C01709=71.781,53.873,81.904,-174.9523,-0.9140,-13823.1111
C01710=77.964,55.051,82.431,-177.5443,-2.1205,-13824.7738
C01711=83.695,52.900,82.857,-179.4162,-1.4469,-13827.7048
C01712=87.788,47.863,83.283,-179.9986,-0.1052,-13831.4003
C01713=90.949,41.570,83.562,-179.9996,-0.0128,-13835.4363
C01714=93.705,34.916,83.562,-179.9986,-0.0127,-13839.5638
C01715=95.920,28.231,83.283,180.0000,-0.1015,-13843.5999
C01716=96.587,21.776,82.857,179.4149,-1.4483,-13847.2948
C01717=94.056,16.202,82.431,177.5455,-2.1207,-13850.2262
C01718=88.851,12.662,81.904,174.9556,-0.9120,-13851.8895
C01719=81.722,11.527,80.892,174.7101,-0.0362,-13851.9713
C01720=73.885,10.553,78.794,175.1749,-0.0294,-13851.8714
C01721=66.709,9.674,75.971,175.9523,-0.0621,-13851.7486
C01722=61.204,8.875,73.167,178.1043,-0.0957,-13851.7492
C01723=57.930,7.507,71.114,-165.0758,11.9424,-13852.6163
C01724=57.039,4.398,70.297,-173.6555,31.1772,-13855.5909
C01725=57.094,1.874,70.261,179.7573,32.5080,-13858.1201
C01726=57.118,0.000,70.285,-180.0000,32.4949,-13860.0000
C01727=57.094,-1.874,70.261,-179.7573,32.5080,-13861.8799
C01728=57.039,-4.398,70.297,173.6555,31.1772,-13864.4091
C01729=57.930,-7.507,71.114,165.0758,11.9424,-13867.3837
C01730=61.204,-8.875,73.167,-178.1043,-0.0957,-13868.2508
C01731=66.709,-9.674,75.971,-175.9523,-0.0621,-13868.2514
C01732=73.885,-10.553,78.794,-175.1749,-0.0294,-13868.1286
C01733=81.722,-11.527,80.892,-174.7101,-0.0362,-13868.0287
C01734=88.851,-12.662,81.904,-174.9556,-0.9120,-13868.1105
C01735=94.056,-16.202,82.431,-177.5455,-2.1207,-13869.7738
C01736=96.587,-21.776,82.857,-179.4149,-1.4483,-13872.7052
C01737=95.920,-28.231,83.283,-180.0000,-0.1015,-13876.4001
C01738=93.705,-34.916,83.562,179.9986,-0.0127,-13880.4362
C01739=90.949,-41.570,83.562,179.9996,-0.0128,-13884.5637
C01740=87.788,-47.863,83.283,179.9986,-0.1052,-13888.5997
C01741=83.695,-52.900,82.857,179.4162,-1.4469,-13892.2952
C01742=77.964,-55.051,82.431,177.5443,-2.1205,-13895.2262
C01743=71.781,-53.873,81.904,174.9523,-0.9140,-13896.8889
C01744=65.937,-49.635,80.892,174.7131,-0.0370,-13896.9711
C01745=59.707,-44.783,78.794,175.1691,-0.0312,-13896.8716
C01746=54.011,-40.330,75.971,175.9514,-0.0603,-13896.7487
C01747=49.553,-37.003,73.167,178.1031,-0.0935,-13896.7500
C01748=46.271,-35.654,71.114,-165.0753,11.9430,-13897.6160
C01749=43.442,-37.223,70.297,-173.6602,31.1794,-13900.5914
C01750=41.697,-39.047,70.261,179.7562,32.5069,-13903.1202
C01751=40.388,-40.388,70.285,-180.0000,32.4978,-13905.0000
C01752=39.047,-41.696,70.261,-179.7558,32.5069,-13906.8791
C01753=37.223,-43.443,70.297,173.6555,31.1756,-13909.4092
C01754=35.654,-46.271,71.114,165.0753,11.9430,-13912.3840
C01755=37.003,-49.553,73.167,-178.1031,-0.0935,-13913.2500
C01756=40.330,-54.011,75.971,-175.9514,-0.0603,-13913.2513
C01757=44.783,-59.707,78.794,-175.1691,-0.0312,-13913.1284
C01758=49.635,-65.937,80.892,-174.7131,-0.0370,-13913.0289
C01759=53.873,-71.781,81.904,-174.9523,-0.9140,-13913.1111
C01760=55.051,-77.964,82.431,-177.5443,-2.1205,-13914.7738
C01761=52.900,-83.695,82.857,-179.4162,-1.4469,-13917.7048
C01762=47.863,-87.788,83.283,-179.9986,-0.1052,-13921.4003
C01763=41.570,-90.949,83.562,-179.9996,-0.0128,-13925.4363
C01764=34.916,-93.705,83.562,-179.9986,-0.0127,-13929.5638
C01765=28.231,-95.920,83.283,180.0000,-0.1015,-13933.5999
C01766=21.776,-96.587,82.857,179.4149,-1.4483,-13937.2948
C01767=16.202,-94.056,82.431,177.5455,-2.1207,-13940.2262
C01768=12.662,-88.851,81.904,174.9556,-0.9120,-13941.8895
C01769=11.527,-81.722,80.892,174.7101,-0.0362,-13941.9713
C01770=10.553,-73.885,78.794,175.1749,-0.0294,-13941.8714
C01771=9.674,-66.709,75.971,175.9523,-0.0621,-13941.7486
C01772=8.875,-61.204,73.167,178.1043,-0.0957,-13941.7492
C01773=7.507,-57.930,71.114,-165.0758,11.9424,-13942.6163
C01774=4.398,-57.039,70.297,-173.6555,31.1772,-13945.5909
C01775=1.874,-57.094,70.261,179.7573,32.5080,-13948.1201
C01776=0.000,-57.118,70.285,-180.0000,32.4949,-13950.0000
C01777=0.000,-57.118,70.285,-180.0000,32.4949,-13950.0000
C01778=-1.874,-57.094,70.261,-179.7573,32.5080,-13951.8799
C01779=-4.398,-57.039,70.297,173.6555,31.1772,-13954.4091
C01780=-7.507,-57.930,71.114,165.0758,11.9424,-13957.3837
C01781=-8.875,-61.204,73.167,-178.1043,-0.0957,-13958.2508
C01782=-9.674,-66.709,75.971,-175.9523,-0.0621,-13958.2514
C01783=-10.553,-73.885,78.794,-175.1749,-0.0294,-13958.1286
C01784=-11.527,-81.722,80.892,-174.7101,-0.0362,-13958.0287
C01785=-12.662,-88.851,81.904,-174.9556,-0.9120,-13958.1105
C01786=-16.202,-94.056,82.431,-177.5455,-2.1207,-13959.7738
C01787=-21.776,-96.587,82.857,-179.4149,-1.4483,-13962.7052
C01788=-28.231,-95.920,83.283,-180.0000,-0.1015,-13966.4001
C01789=-34.916,-93.705,83.562,179.9986,-0.0127,-13970.4362
C01790=-41.570,-90.949,83.562,179.9996,-0.0128,-13974.5637
C01791=-47.863,-87.788,83.283,179.9986,-0.1052,-13978.5997
C01792=-52.900,-83.695,82.857,179.4162,-1.4469,-13982.2952
C01793=-55.051,-77.964,82.431,177.5443,-2.1205,-13985.2262
C01794=-53.873,-71.781,81.904,174.9523,-0.9140,-13986.8889
C01795=-49.635,-65.937,80.892,174.7131,-0.0370,-13986.9711
C01796=-44.783,-59.707,78.794,175.1691,-0.0312,-13986.8716
C01797=-40.330,-54.011,75.971,175.9514,-0.0603,-13986.7487
C01798=-37.003,-49.553,73.167,178.1031,-0.0935,-13986.7500
C01799=-35.654,-46.271,71.114,-165.0753,11.9430,-13987.6160
C01800=-37.223,-43.442,70.297,-173.6602,31.1794,-13990.5914
C01801=-39.047,-41.697,70.261,179.7562,32.5069,-13993.1202
C01802=-40.388,-40.388,70.285,-180.0000,32.4978,-13995.0000
C01803=-41.696,-39.047,70.261,-179.7558,32.5069,-13996.8791
C01804=-43.443,-37.223,70.297,173.6555,31.1756,-13999.4092
C01805=-46.271,-35.654,71.114,165.0753,11.9430,-14002.3840
C01806=-49.553,-37.003,73.167,-178.1031,-0.0935,-14003.2500
C01807=-54.011,-40.330,75.971,-175.9514,-0.0603,-14003.2513
C01808=-59.707,-44.783,78.794,-175.1691,-0.0312,-14003.1284
C01809=-65.937,-49.635,80.892,-174.7131,-0.0370,-14003.0289
C01810=-71.781,-53.873,81.904,-174.9523,-0.9140,-14003.1111
C01811=-77.964,-55.051,82.431,-177.5443,-2.1205,-14004.7738
C01812=-83.695,-52.900,82.857,-179.4162,-1.4469,-14007.7048
C01813=-87.788,-47.863,83.283,-179.9986,-0.1052,-14011.4003
C01814=-90.949,-41.570,83.562,-179.9996,-0.0128,-14015.4363
C01815=-93.705,-34.916,83.562,-179.9986,-0.0127,-14019.5638
C01816=-95.920,-28.231,83.283,180.0000,-0.1015,-14023.5999
C01817=-96.587,-21.776,82.857,179.4149,-1.4483,-14027.2948
C01818=-94.056,-16.202,82.431,177.5455,-2.1207,-14030.2262
C01819=-88.851,-12.662,81.904,174.9556,-0.9120,-14031.8895
C01820=-81.722,-11.527,80.892,174.7101,-0.0362,-14031.9713
C01821=-73.885,-10.553,78.794,175.1749,-0.0294,-14031.8714
C01822=-66.709,-9.674,75.971,175.9523,-0.0621,-14031.7486
C01823=-61.204,-8.875,73.167,178.1043,-0.0957,-14031.7492
C01824=-57.930,-7.507,71.114,-165.0758,11.9424,-14032.6163
C01825=-57.039,-4.398,70.297,-173.6555,31.1772,-14035.5909
C01826=-57.094,-1.874,70.261,179.7573,32.5080,-14038.1201
C01827=-57.118,0.000,70.285,-180.0000,32.4949,-14040.0000
C01828=-57.094,1.874,70.261,-179.7573,32.5080,-14041.8799
C01829=-57.039,4.398,70.297,173.6555,31.1772,-14044.4091
C01830=-57.930,7.507,71.114,165.0758,11.9424,-14047.3837
C01831=-61.204,8.875,73.167,-178.1043,-0.0957,-14048.2508
C01832=-66.709,9.674,75.971,-175.9523,-0.0621,-14048.2514
C01833=-73.885,10.553,78.794,-175.1749,-0.0294,-14048.1286
C01834=-81.722,11.527,80.892,-174.7101,-0.0362,-14048.0287
C01835=-88.851,12.662,81.904,-174.9556,-0.9120,-14048.1105
C01836=-94.056,16.202,82.431,-177.5455,-2.1207,-14049.7738
C01837=-96.587,21.776,82.857,-179.4149,-1.4483,-14052.7052
C01838=-95.920,28.231,83.283,-180.0000,-0.1015,-14056.4001
C01839=-93.705,34.916,83.562,179.9986,-0.0127,-14060.4362
C01840=-90.949,41.570,83.562,179.9996,-0.0128,-14064.5637
C01841=-87.788,47.863,83.283,179.9986,-0.1052,-14068.5997
C01842=-83.695,52.900,82.857,179.4162,-1.4469,-14072.2952
C01843=-77.964,55.051,82.431,177.5443,-2.1205,-14075.2262
C01844=-71.781,53.873,81.904,174.9523,-0.9140,-14076.8889
C01845=-65.937,49.635,80.892,174.7131,-0.0370,-14076.9711
C01846=-59.707,44.783,78.794,175.1691,-0.0312,-14076.8716
C01847=-54.011,40.330,75.971,175.9514,-0.0603,-14076.7487
C01848=-49.553,37.003,73.167,178.1031,-0.0935,-14076.7500
C01849=-46.271,35.654,71.114,-165.0753,11.9430,-14077.6160
C01850=-43.442,37.223,70.297,-173.6602,31.1794,-14080.5914
C01851=-41.697,39.047,70.261,179.7562,32.5069,-14083.1202
C01852=-40.388,40.388,70.285,180.0000,32.4978,-14085.0000
C01853=-39.047,41.696,70.261,-179.7558,32.5069,-14086.8791
C01854=-37.223,43.443,70.297,173.6555,31.1756,-14089.4092
C01855=-35.654,46.271,71.114,165.0753,11.9430,-14092.3840
C01856=-37.003,49.553,73.167,-178.1031,-0.0935,-14093.2500
C01857=-40.330,54.011,75.971,-175.9514,-0.0603,-14093.2513
C01858=-44.783,59.707,78.794,-175.1691,-0.0312,-14093.1284
C01859=-49.635,65.937,80.892,-174.7131,-0.0370,-14093.0289
C01860=-53.873,71.781,81.904,-174.9523,-0.9140,-14093.1111
C01861=-55.051,77.964,82.431,-177.5443,-2.1205,-14094.7738
C01862=-52.900,83.695,82.857,-179.4162,-1.4469,-14097.7048
C01863=-47.863,87.788,83.283,-179.9986,-0.1052,-14101.4003
C01864=-41.570,90.949,83.562,-179.9996,-0.0128,-14105.4363
C01865=-34.916,93.705,83.562,-179.9986,-0.0127,-14109.5638
C01866=-28.231,95.920,83.283,180.0000,-0.1015,-14113.5999
C01867=-21.776,96.587,82.857,179.4149,-1.4483,-14117.2948
C01868=-16.202,94.056,82.431,177.5455,-2.1207,-14120.2262
C01869=-12.662,88.851,81.904,174.9556,-0.9120,-14121.8895
C01870=-11.527,81.722,80.892,174.7101,-0.0362,-14121.9713
C01871=-10.553,73.885,78.794,175.1749,-0.0294,-14121.8714
C01872=-9.674,66.709,75.971,175.9523,-0.0621,-14121.7486
C01873=-8.875,61.204,73.167,178.1043,-0.0957,-14121.7492
C01874=-7.507,57.930,71.114,-165.0758,11.9424,-14122.6163
C01875=-4.398,57.039,70.297,-173.6555,31.1772,-14125.5909
C01876=-1.874,57.094,70.261,179.7573,32.5080,-14128.1201
C01877=0.000,57.118,70.285,180.0000,32.4949,-14130.0000
C01878=0.000,55.957,72.154,180.0000,31.1976,-14130.0000
C01879=1.768,55.936,72.129,-179.7768,31.2086,-14131.8104
C01880=4.219,55.892,72.166,173.7293,29.8078,-14134.3168
C01881=7.293,56.844,73.015,166.0480,10.7254,-14137.3110
C01882=8.627,60.270,75.143,-177.9267,-0.0854,-14138.1459
C01883=9.417,65.995,78.036,-176.1598,-0.0428,-14138.1209
C01884=10.308,73.408,80.927,-175.6017,-0.0195,-14137.9932
C01885=11.295,81.446,83.062,-175.3181,-0.0225,-14137.8955
C01886=12.427,88.723,84.088,-175.5876,-0.7793,-14137.9733
C01887=15.989,94.030,84.621,-177.8561,-1.8342,-14139.6504
C01888=21.612,96.617,85.050,-179.4972,-1.2499,-14142.6088
C01889=28.131,95.953,85.481,-179.9978,-0.0889,-14146.3398
C01890=34.883,93.717,85.762,179.9986,-0.0127,-14150.4161
C01891=41.602,90.934,85.762,179.9996,-0.0128,-14154.5839
C01892=47.957,87.741,85.481,-179.9995,-0.0846,-14158.6599
C01893=53.037,83.601,85.050,179.4963,-1.2492,-14162.3913
C01894=55.184,77.795,84.621,177.8577,-1.8362,-14165.3500
C01895=53.949,71.524,84.088,175.5865,-0.7799,-14167.0265
C01896=49.604,65.578,83.062,175.3163,-0.0261,-14167.1043
C01897=44.618,59.196,80.927,175.6070,-0.0220,-14167.0066
C01898=40.007,53.324,78.036,176.1608,-0.0420,-14166.8795
C01899=36.517,48.718,75.143,177.9288,-0.0843,-14166.8537
C01900=35.037,45.351,73.015,-166.0442,10.7217,-14167.6887
C01901=36.538,42.505,72.166,-173.7278,29.8093,-14170.6829
C01902=38.303,40.803,72.129,179.7748,31.2094,-14173.1899
C01903=39.567,39.567,72.154,180.0000,31.1989,-14175.0000
C01904=40.803,38.303,72.129,-179.7748,31.2094,-14176.8101
C01905=42.506,36.538,72.166,173.7274,29.8092,-14179.3178
C01906=45.352,35.037,73.015,166.0441,10.7215,-14182.3119
C01907=48.718,36.517,75.143,-177.9288,-0.0843,-14183.1463
C01908=53.324,40.007,78.036,-176.1608,-0.0420,-14183.1205
C01909=59.196,44.618,80.927,-175.6070,-0.0220,-14182.9934
C01910=65.578,49.604,83.062,-175.3163,-0.0261,-14182.8957
C01911=71.524,53.949,84.088,-175.5865,-0.7799,-14182.9735
C01912=77.795,55.184,84.621,-177.8577,-1.8362,-14184.6500
C01913=83.601,53.037,85.050,-179.4963,-1.2492,-14187.6087
C01914=87.741,47.957,85.481,179.9995,-0.0846,-14191.3401
C01915=90.934,41.602,85.762,-179.9996,-0.0128,-14195.4161
C01916=93.717,34.883,85.762,-179.9986,-0.0127,-14199.5839
C01917=95.953,28.131,85.481,179.9978,-0.0889,-14203.6602
C01918=96.617,21.612,85.050,179.4972,-1.2499,-14207.3912
C01919=94.030,15.989,84.621,177.8561,-1.8342,-14210.3496
C01920=88.723,12.427,84.088,175.5876,-0.7793,-14212.0267
C01921=81.446,11.295,83.062,175.3181,-0.0225,-14212.1045
C01922=73.408,10.308,80.927,175.6017,-0.0195,-14212.0068
C01923=65.995,9.417,78.036,176.1598,-0.0428,-14211.8791
C01924=60.270,8.627,75.143,177.9267,-0.0854,-14211.8541
C01925=56.844,7.293,73.015,-166.0480,10.7254,-14212.6890
C01926=55.892,4.219,72.166,-173.7293,29.8078,-14215.6832
C01927=55.936,1.768,72.129,179.7768,31.2086,-14218.1896
C01928=55.957,0.000,72.154,180.0000,31.1976,-14220.0000
C01929=55.936,-1.767,72.129,-179.7762,31.2086,-14221.8094
C01930=55.892,-4.220,72.166,173.7222,29.8074,-14224.3178
C01931=56.844,-7.293,73.015,166.0480,10.7254,-14227.3110
C01932=60.270,-8.627,75.143,-177.9267,-0.0854,-14228.1459
C01933=65.995,-9.417,78.036,-176.1598,-0.0428,-14228.1209
C01934=73.408,-10.308,80.927,-175.6017,-0.0195,-14227.9932
C01935=81.446,-11.295,83.062,-175.3181,-0.0225,-14227.8955
C01936=88.723,-12.427,84.088,-175.5876,-0.7793,-14227.9733
C01937=94.030,-15.989,84.621,-177.8561,-1.8342,-14229.6504
C01938=96.617,-21.612,85.050,-179.4972,-1.2499,-14232.6088
C01939=95.953,-28.131,85.481,-179.9978,-0.0889,-14236.3398
C01940=93.717,-34.883,85.762,179.9986,-0.0127,-14240.4161
C01941=90.934,-41.602,85.762,179.9996,-0.0128,-14244.5839
C01942=87.741,-47.957,85.481,-179.9995,-0.0846,-14248.6599
C01943=83.601,-53.037,85.050,179.4963,-1.2492,-14252.3913
C01944=77.795,-55.184,84.621,177.8577,-1.8362,-14255.3500
C01945=71.524,-53.949,84.088,175.5865,-0.7799,-14257.0265
C01946=65.578,-49.604,83.062,175.3163,-0.0261,-14257.1043
C01947=59.196,-44.618,80.927,175.6070,-0.0220,-14257.0066
C01948=53.324,-40.007,78.036,176.1608,-0.0420,-14256.8795
C01949=48.718,-36.517,75.143,177.9288,-0.0843,-14256.8537
C01950=45.351,-35.037,73.015,-166.0442,10.7217,-14257.6887
C01951=42.505,-36.538,72.166,-173.7278,29.8093,-14260.6829
C01952=40.803,-38.303,72.129,179.7748,31.2094,-14263.1899
C01953=39.567,-39.567,72.154,-180.0000,31.1989,-14265.0000
C01954=38.303,-40.803,72.129,-179.7748,31.2094,-14266.8101
C01955=36.538,-42.506,72.166,173.7274,29.8092,-14269.3178
C01956=35.037,-45.352,73.015,166.0441,10.7215,-14272.3119
C01957=36.517,-48.718,75.143,-177.9288,-0.0843,-14273.1463
C01958=40.007,-53.324,78.036,-176.1608,-0.0420,-14273.1205
C01959=44.618,-59.196,80.927,-175.6070,-0.0220,-14272.9934
C01960=49.604,-65.578,83.062,-175.3163,-0.0261,-14272.8957
C01961=53.949,-71.524,84.088,-175.5865,-0.7799,-14272.9735
C01962=55.184,-77.795,84.621,-177.8577,-1.8362,-14274.6500
C01963=53.037,-83.601,85.050,-179.4963,-1.2492,-14277.6087
C01964=47.957,-87.741,85.481,179.9995,-0.0846,-14281.3401
C01965=41.602,-90.934,85.762,-179.9996,-0.0128,-14285.4161
C01966=34.883,-93.717,85.762,-179.9986,-0.0127,-14289.5839
C01967=28.131,-95.953,85.481,179.9978,-0.0889,-14293.6602
C01968=21.612,-96.617,85.050,179.4972,-1.2499,-14297.3912
C01969=15.989,-94.030,84.621,177.8561,-1.8342,-14300.3496
C01970=12.427,-88.723,84.088,175.5876,-0.7793,-14302.0267
C01971=11.295,-81.446,83.062,175.3181,-0.0225,-14302.1045
C01972=10.308,-73.408,80.927,175.6017,-0.0195,-14302.0068
C01973=9.417,-65.995,78.036,176.1598,-0.0428,-14301.8791
C01974=8.627,-60.270,75.143,177.9267,-0.0854,-14301.8541
C01975=7.293,-56.844,73.015,-166.0480,10.7254,-14302.6890
C01976=4.219,-55.892,72.166,-173.7293,29.8078,-14305.6832
C01977=1.768,-55.936,72.129,179.7768,31.2086,-14308.1896
C01978=0.000,-55.957,72.154,-180.0000,31.1976,-14310.0000
C01979=0.000,-55.957,72.154,-180.0000,31.1976,-14310.0000
C01980=-1.767,-55.936,72.129,-179.7762,31.2086,-14311.8094
C01981=-4.220,-55.892,72.166,173.7222,29.8074,-14314.3178
C01982=-7.293,-56.844,73.015,166.0480,10.7254,-14317.3110
C01983=-8.627,-60.270,75.143,-177.9267,-0.0854,-14318.1459
C01984=-9.417,-65.995,78.036,-176.1598,-0.0428,-14318.1209
C01985=-10.308,-73.408,80.927,-175.6017,-0.0195,-14317.9932
C01986=-11.295,-81.446,83.062,-175.3181,-0.0225,-14317.8955
C01987=-12.427,-88.723,84.088,-175.5876,-0.7793,-14317.9733
C01988=-15.989,-94.030,84.621,-177.8561,-1.8342,-14319.6504
C01989=-21.612,-96.617,85.050,-179.4972,-1.2499,-14322.6088
C01990=-28.131,-95.953,85.481,-179.9978,-0.0889,-14326.3398
C01991=-34.883,-93.717,85.762,179.9986,-0.0127,-14330.4161
C01992=-41.602,-90.934,85.762,179.9996,-0.0128,-14334.5839
C01993=-47.957,-87.741,85.481,-179.9995,-0.0846,-14338.6599
C01994=-53.037,-83.601,85.050,179.4963,-1.2492,-14342.3913
C01995=-55.184,-77.795,84.621,177.8577,-1.8362,-14345.3500
C01996=-53.949,-71.524,84.088,175.5865,-0.7799,-14347.0265
C01997=-49.604,-65.578,83.062,175.3163,-0.0261,-14347.1043
C01998=-44.618,-59.196,80.927,175.6070,-0.0220,-14347.0066
C01999=-40.007,-53.324,78.036,176.1608,-0.0420,-14346.8795
///TOOL 0
///POSTYPE ANGLE
///ANGLE
EC00000=0.0000,10788.4794
EC00001=0.0000,10790.0243
EC00002=0.0000,10790.2854
EC00003=0.0000,10790.3475
EC00004=0.0000,10790.4499
EC00005=0.0000,10790.8103
EC00006=0.0000,10792.0037
EC00007=0.0000,10794.8371
EC00008=0.0000,10797.5483
EC00009=0.0000,10800.0000
EC00010=0.0000,10802.4517
EC00011=0.0000,10805.1629
EC00012=0.0000,10807.9963
EC00013=0.0000,10809.1897
EC00014=0.0000,10809.5501
EC00015=0.0000,10809.6525
EC00016=0.0000,10809.7146
EC00017=0.0000,10809.9757
EC00018=0.0000,10811.5206
EC00019=0.0000,10814.1038
EC00020=0.0000,10817.2974
EC00021=0.0000,10820.7433
EC00022=0.0000,10824.2566
EC00023=0.0000,10827.7026
EC00024=0.0000,10830.8962
EC00025=0.0000,10833.4793
EC00026=0.0000,10835.0245
EC00027=0.0000,10835.2855
EC00028=0.0000,10835.3476
EC00029=0.0000,10835.4495
EC00030=0.0000,10835.8105
EC00031=0.0000,10837.0038
EC00032=0.0000,10839.8372
EC00033=0.0000,10842.5482
EC00034=0.0000,10845.0000
EC00035=0.0000,10847.4518
EC00036=0.0000,10850.1628
EC00037=0.0000,10852.9966
EC00038=0.0000,10854.1895
EC00039=0.0000,10854.5505
EC00040=0.0000,10854.6524
EC00041=0.0000,10854.7145
EC00042=0.0000,10854.9755
EC00043=0.0000,10856.5207
EC00044=0.0000,10859.1038
EC00045=0.0000,10862.2974
EC00046=0.0000,10865.7434
EC00047=0.0000,10869.2567
EC00048=0.0000,10872.7026
EC00049=0.0000,10875.8962
EC00050=0.0000,10878.4794
EC00051=0.0000,10880.0243
EC00052=0.0000,10880.2854
EC00053=0.0000,10880.3475
EC00054=0.0000,10880.4499
EC00055=0.0000,10880.8103
EC00056=0.0000,10882.0037
EC00057=0.0000,10884.8371
EC00058=0.0000,10887.5483
EC00059=0.0000,10890.0000
EC00060=0.0000,10890.0000
EC00061=0.0000,10892.3954
EC00062=0.0000,10895.0881
EC00063=0.0000,10897.9350
EC00064=0.0000,10899.0911
EC00065=0.0000,10899.4060
EC00066=0.0000,10899.4709
EC00067=0.0000,10899.5004
EC00068=0.0000,10899.7298
EC00069=0.0000,10901.2851
EC00070=0.0000,10903.9122
EC00071=0.0000,10907.1736
EC00072=0.0000,10910.7008
EC00073=0.0000,10914.2992
EC00074=0.0000,10917.8267
EC00075=0.0000,10921.0877
EC00076=0.0000,10923.7152
EC00077=0.0000,10925.2699
EC00078=0.0000,10925.4993
EC00079=0.0000,10925.5293
EC00080=0.0000,10925.5938
EC00081=0.0000,10925.9087
EC00082=0.0000,10927.0654
EC00083=0.0000,10929.9123
EC00084=0.0000,10932.6047
EC00085=0.0000,10935.0000
EC00086=0.0000,10937.3953
EC00087=0.0000,10940.0883
EC00088=0.0000,10942.9346
EC00089=0.0000,10944.0913
EC00090=0.0000,10944.4062
EC00091=0.0000,10944.4707
EC00092=0.0000,10944.5007
EC00093=0.0000,10944.7301
EC00094=0.0000,10946.2848
EC00095=0.0000,10948.9123
EC00096=0.0000,10952.1733
EC00097=0.0000,10955.7008
EC00098=0.0000,10959.2992
EC00099=0.0000,10962.8264
EC00100=0.0000,10966.0878
EC00101=0.0000,10968.7149
EC00102=0.0000,10970.2702
EC00103=0.0000,10970.4996
EC00104=0.0000,10970.5291
EC00105=0.0000,10970.5940
EC00106=0.0000,10970.9089
EC00107=0.0000,10972.0650
EC00108=0.0000,10974.9119
EC00109=0.0000,10977.6046
EC00110=0.0000,10980.0000
EC00111=0.0000,10982.3954
EC00112=0.0000,10985.0881
EC00113=0.0000,10987.9350
EC00114=0.0000,10989.0911
EC00115=0.0000,10989.4060
EC00116=0.0000,10989.4709
EC00117=0.0000,10989.5004
EC00118=0.0000,10989.7298
EC00119=0.0000,10991.2851
EC00120=0.0000,10993.9122
EC00121=0.0000,10997.1736
EC00122=0.0000,11000.7008
EC00123=0.0000,11004.2992
EC00124=0.0000,11007.8267
EC00125=0.0000,11011.0877
EC00126=0.0000,11013.7152
EC00127=0.0000,11015.2699
EC00128=0.0000,11015.4993
EC00129=0.0000,11015.5293
EC00130=0.0000,11015.5938
EC00131=0.0000,11015.9087
EC00132=0.0000,11017.0654
EC00133=0.0000,11019.9123
EC00134=0.0000,11022.6047
EC00135=0.0000,11025.0000
EC00136=0.0000,11027.3953
EC00137=0.0000,11030.0883
EC00138=0.0000,11032.9346
EC00139=0.0000,11034.0913
EC00140=0.0000,11034.4062
EC00141=0.0000,11034.4707
EC00142=0.0000,11034.5007
EC00143=0.0000,11034.7301
EC00144=0.0000,11036.2848
EC00145=0.0000,11038.9123
EC00146=0.0000,11042.1733
EC00147=0.0000,11045.7008
EC00148=0.0000,11049.2992
EC00149=0.0000,11052.8264
EC00150=0.0000,11056.0878
EC00151=0.0000,11058.7149
EC00152=0.0000,11060.2702
EC00153=0.0000,11060.4996
EC00154=0.0000,11060.5291
EC00155=0.0000,11060.5940
EC00156=0.0000,11060.9089
EC00157=0.0000,11062.0650
EC00158=0.0000,11064.9119
EC00159=0.0000,11067.6046
EC00160=0.0000,11070.0000
EC00161=0.0000,11070.0000
EC00162=0.0000,11072.3954
EC00163=0.0000,11075.0881
EC00164=0.0000,11077.9350
EC00165=0.0000,11079.0911
EC00166=0.0000,11079.4060
EC00167=0.0000,11079.4709
EC00168=0.0000,11079.5004
EC00169=0.0000,11079.7298
EC00170=0.0000,11081.2851
EC00171=0.0000,11083.9122
EC00172=0.0000,11087.1736
EC00173=0.0000,11090.7008
EC00174=0.0000,11094.2992
EC00175=0.0000,11097.8267
EC00176=0.0000,11101.0877
EC00177=0.0000,11103.7152
EC00178=0.0000,11105.2699
EC00179=0.0000,11105.4993
EC00180=0.0000,11105.5293
EC00181=0.0000,11105.5938
EC00182=0.0000,11105.9087
EC00183=0.0000,11107.0654
EC00184=0.0000,11109.9123
EC00185=0.0000,11112.6047
EC00186=0.0000,11115.0000
EC00187=0.0000,11117.3953
EC00188=0.0000,11120.0883
EC00189=0.0000,11122.9346
EC00190=0.0000,11124.0913
EC00191=0.0000,11124.4062
EC00192=0.0000,11124.4707
EC00193=0.0000,11124.5007
EC00194=0.0000,11124.7301
EC00195=0.0000,11126.2848
EC00196=0.0000,11128.9123
EC00197=0.0000,11132.1733
EC00198=0.0000,11135.7008
EC00199=0.0000,11139.2992
EC00200=0.0000,11142.8264
EC00201=0.0000,11146.0878
EC00202=0.0000,11148.7149
EC00203=0.0000,11150.2702
EC00204=0.0000,11150.4996
EC00205=0.0000,11150.5291
EC00206=0.0000,11150.5940
EC00207=0.0000,11150.9089
EC00208=0.0000,11152.0650
EC00209=0.0000,11154.9119
EC00210=0.0000,11157.6046
EC00211=0.0000,11160.0000
EC00212=0.0000,11162.3954
EC00213=0.0000,11165.0881
EC00214=0.0000,11167.9350
EC00215=0.0000,11169.0911
EC00216=0.0000,11169.4060
EC00217=0.0000,11169.4709
EC00218=0.0000,11169.5004
EC00219=0.0000,11169.7298
EC00220=0.0000,11171.2851
EC00221=0.0000,11173.9122
EC00222=0.0000,11177.1736
EC00223=0.0000,11180.7008
EC00224=0.0000,11184.2992
EC00225=0.0000,11187.8267
EC00226=0.0000,11191.0877
EC00227=0.0000,11193.7152
EC00228=0.0000,11195.2699
EC00229=0.0000,11195.4993
EC00230=0.0000,11195.5293
EC00231=0.0000,11195.5938
EC00232=0.0000,11195.9087
EC00233=0.0000,11197.0654
EC00234=0.0000,11199.9123
EC00235=0.0000,11202.6047
EC00236=0.0000,11205.0000
EC00237=0.0000,11207.3953
EC00238=0.0000,11210.0883
EC00239=0.0000,11212.9346
EC00240=0.0000,11214.0913
EC00241=0.0000,11214.4062
EC00242=0.0000,11214.4707
EC00243=0.0000,11214.5007
EC00244=0.0000,11214.7301
EC00245=0.0000,11216.2848
EC00246=0.0000,11218.9123
EC00247=0.0000,11222.1733
EC00248=0.0000,11225.7008
EC00249=0.0000,11229.2992
EC00250=0.0000,11232.8264
EC00251=0.0000,11236.0878
EC00252=0.0000,11238.7149
EC00253=0.0000,11240.2702
EC00254=0.0000,11240.4996
EC00255=0.0000,11240.5291
EC00256=0.0000,11240.5940
EC00257=0.0000,11240.9089
EC00258=0.0000,11242.0650
EC00259=0.0000,11244.9119
EC00260=0.0000,11247.6046
EC00261=0.0000,11250.0000
EC00262=0.0000,11250.0000
EC00263=0.0000,11252.3363
EC00264=0.0000,11255.0104
EC00265=0.0000,11257.8714
EC00266=0.0000,11258.9912
EC00267=0.0000,11259.2604
EC00268=0.0000,11259.2892
EC00269=0.0000,11259.2905
EC00270=0.0000,11259.4907
EC00271=0.0000,11261.0568
EC00272=0.0000,11263.7273
EC00273=0.0000,11267.0541
EC00274=0.0000,11270.6599
EC00275=0.0000,11274.3400
EC00276=0.0000,11277.9461
EC00277=0.0000,11281.2727
EC00278=0.0000,11283.9430
EC00279=0.0000,11285.5096
EC00280=0.0000,11285.7099
EC00281=0.0000,11285.7103
EC00282=0.0000,11285.7399
EC00283=0.0000,11286.0092
EC00284=0.0000,11287.1289
EC00285=0.0000,11289.9895
EC00286=0.0000,11292.6632
EC00287=0.0000,11295.0000
EC00288=0.0000,11297.3362
EC00289=0.0000,11300.0105
EC00290=0.0000,11302.8711
EC00291=0.0000,11303.9908
EC00292=0.0000,11304.2601
EC00293=0.0000,11304.2897
EC00294=0.0000,11304.2901
EC00295=0.0000,11304.4904
EC00296=0.0000,11306.0570
EC00297=0.0000,11308.7273
EC00298=0.0000,11312.0539
EC00299=0.0000,11315.6600
EC00300=0.0000,11319.3401
EC00301=0.0000,11322.9459
EC00302=0.0000,11326.2727
EC00303=0.0000,11328.9432
EC00304=0.0000,11330.5093
EC00305=0.0000,11330.7095
EC00306=0.0000,11330.7108
EC00307=0.0000,11330.7396
EC00308=0.0000,11331.0088
EC00309=0.0000,11332.1286
EC00310=0.0000,11334.9896
EC00311=0.0000,11337.6637
EC00312=0.0000,11340.0000
EC00313=0.0000,11342.3363
EC00314=0.0000,11345.0112
EC00315=0.0000,11347.8714
EC00316=0.0000,11348.9912
EC00317=0.0000,11349.2604
EC00318=0.0000,11349.2892
EC00319=0.0000,11349.2905
EC00320=0.0000,11349.4907
EC00321=0.0000,11351.0568
EC00322=0.0000,11353.7273
EC00323=0.0000,11357.0541
EC00324=0.0000,11360.6599
EC00325=0.0000,11364.3400
EC00326=0.0000,11367.9461
EC00327=0.0000,11371.2727
EC00328=0.0000,11373.9430
EC00329=0.0000,11375.5096
EC00330=0.0000,11375.7099
EC00331=0.0000,11375.7103
EC00332=0.0000,11375.7399
EC00333=0.0000,11376.0092
EC00334=0.0000,11377.1289
EC00335=0.0000,11379.9895
EC00336=0.0000,11382.6632
EC00337=0.0000,11385.0000
EC00338=0.0000,11387.3362
EC00339=0.0000,11390.0105
EC00340=0.0000,11392.8711
EC00341=0.0000,11393.9908
EC00342=0.0000,11394.2601
EC00343=0.0000,11394.2897
EC00344=0.0000,11394.2901
EC00345=0.0000,11394.4904
EC00346=0.0000,11396.0570
EC00347=0.0000,11398.7273
EC00348=0.0000,11402.0539
EC00349=0.0000,11405.6600
EC00350=0.0000,11409.3401
EC00351=0.0000,11412.9459
EC00352=0.0000,11416.2727
EC00353=0.0000,11418.9432
EC00354=0.0000,11420.5093
EC00355=0.0000,11420.7095
EC00356=0.0000,11420.7108
EC00357=0.0000,11420.7396
EC00358=0.0000,11421.0088
EC00359=0.0000,11422.1286
EC00360=0.0000,11424.9896
EC00361=0.0000,11427.6637
EC00362=0.0000,11430.0000
EC00363=0.0000,11430.0000
EC00364=0.0000,11432.3363
EC00365=0.0000,11435.0112
EC00366=0.0000,11437.8714
EC00367=0.0000,11438.9912
EC00368=0.0000,11439.2604
EC00369=0.0000,11439.2892
EC00370=0.0000,11439.2905
EC00371=0.0000,11439.4907
EC00372=0.0000,11441.0568
EC00373=0.0000,11443.7273
EC00374=0.0000,11447.0541
EC00375=0.0000,11450.6599
EC00376=0.0000,11454.3400
EC00377=0.0000,11457.9461
EC00378=0.0000,11461.2727
EC00379=0.0000,11463.9430
EC00380=0.0000,11465.5096
EC00381=0.0000,11465.7099
EC00382=0.0000,11465.7103
EC00383=0.0000,11465.7399
EC00384=0.0000,11466.0092
EC00385=0.0000,11467.1289
EC00386=0.0000,11469.9895
EC00387=0.0000,11472.6632
EC00388=0.0000,11475.0000
EC00389=0.0000,11477.3362
EC00390=0.0000,11480.0105
EC00391=0.0000,11482.8711
EC00392=0.0000,11483.9908
EC00393=0.0000,11484.2601
EC00394=0.0000,11484.2897
EC00395=0.0000,11484.2901
EC00396=0.0000,11484.4904
EC00397=0.0000,11486.0570
EC00398=0.0000,11488.7273
EC00399=0.0000,11492.0539
EC00400=0.0000,11495.6600
EC00401=0.0000,11499.3401
EC00402=0.0000,11502.9459
EC00403=0.0000,11506.2727
EC00404=0.0000,11508.9432
EC00405=0.0000,11510.5093
EC00406=0.0000,11510.7095
EC00407=0.0000,11510.7108
EC00408=0.0000,11510.7396
EC00409=0.0000,11511.0088
EC00410=0.0000,11512.1286
EC00411=0.0000,11514.9896
EC00412=0.0000,11517.6637
EC00413=0.0000,11520.0000
EC00414=0.0000,11522.3363
EC00415=0.0000,11525.0112
EC00416=0.0000,11527.8714
EC00417=0.0000,11528.9912
EC00418=0.0000,11529.2604
EC00419=0.0000,11529.2892
EC00420=0.0000,11529.2905
EC00421=0.0000,11529.4907
EC00422=0.0000,11531.0568
EC00423=0.0000,11533.7273
EC00424=0.0000,11537.0541
EC00425=0.0000,11540.6599
EC00426=0.0000,11544.3400
EC00427=0.0000,11547.9461
EC00428=0.0000,11551.2727
EC00429=0.0000,11553.9430
EC00430=0.0000,11555.5096
EC00431=0.0000,11555.7099
EC00432=0.0000,11555.7103
EC00433=0.0000,11555.7399
EC00434=0.0000,11556.0092
EC00435=0.0000,11557.1289
EC00436=0.0000,11559.9895
EC00437=0.0000,11562.6632
EC00438=0.0000,11565.0000
EC00439=0.0000,11567.3362
EC00440=0.0000,11570.0105
EC00441=0.0000,11572.8711
EC00442=0.0000,11573.9908
EC00443=0.0000,11574.2601
EC00444=0.0000,11574.2897
EC00445=0.0000,11574.2901
EC00446=0.0000,11574.4904
EC00447=0.0000,11576.0570
EC00448=0.0000,11578.7273
EC00449=0.0000,11582.0539
EC00450=0.0000,11585.6600
EC00451=0.0000,11589.3401
EC00452=0.0000,11592.9459
EC00453=0.0000,11596.2727
EC00454=0.0000,11598.9432
EC00455=0.0000,11600.5093
EC00456=0.0000,11600.7095
EC00457=0.0000,11600.7108
EC00458=0.0000,11600.7396
EC00459=0.0000,11601.0088
EC00460=0.0000,11602.1286
EC00461=0.0000,11604.9888
EC00462=0.0000,11607.6637
EC00463=0.0000,11610.0000
EC00464=0.0000,11610.0000
EC00465=0.0000,11612.2761
EC00466=0.0000,11614.9310
EC00467=0.0000,11617.8063
EC00468=0.0000,11618.8881
EC00469=0.0000,11619.1126
EC00470=0.0000,11619.1102
EC00471=0.0000,11619.0849
EC00472=0.0000,11619.2589
EC00473=0.0000,11620.8371
EC00474=0.0000,11623.5503
EC00475=0.0000,11626.9400
EC00476=0.0000,11630.6205
EC00477=0.0000,11634.3795
EC00478=0.0000,11638.0601
EC00479=0.0000,11641.4498
EC00480=0.0000,11644.1627
EC00481=0.0000,11645.7411
EC00482=0.0000,11645.9150
EC00483=0.0000,11645.8901
EC00484=0.0000,11645.8871
EC00485=0.0000,11646.1114
EC00486=0.0000,11647.1942
EC00487=0.0000,11650.0690
EC00488=0.0000,11652.7235
EC00489=0.0000,11655.0000
EC00490=0.0000,11657.2759
EC00491=0.0000,11659.9310
EC00492=0.0000,11662.8058
EC00493=0.0000,11663.8886
EC00494=0.0000,11664.1129
EC00495=0.0000,11664.1099
EC00496=0.0000,11664.0850
EC00497=0.0000,11664.2589
EC00498=0.0000,11665.8373
EC00499=0.0000,11668.5502
EC00500=0.0000,11671.9399
EC00501=0.0000,11675.6205
EC00502=0.0000,11679.3795
EC00503=0.0000,11683.0600
EC00504=0.0000,11686.4497
EC00505=0.0000,11689.1629
EC00506=0.0000,11690.7411
EC00507=0.0000,11690.9151
EC00508=0.0000,11690.8898
EC00509=0.0000,11690.8874
EC00510=0.0000,11691.1119
EC00511=0.0000,11692.1937
EC00512=0.0000,11695.0690
EC00513=0.0000,11697.7239
EC00514=0.0000,11700.0000
EC00515=0.0000,11702.2761
EC00516=0.0000,11704.9310
EC00517=0.0000,11707.8063
EC00518=0.0000,11708.8881
EC00519=0.0000,11709.1126
EC00520=0.0000,11709.1102
EC00521=0.0000,11709.0849
EC00522=0.0000,11709.2589
EC00523=0.0000,11710.8371
EC00524=0.0000,11713.5503
EC00525=0.0000,11716.9400
EC00526=0.0000,11720.6205
EC00527=0.0000,11724.3795
EC00528=0.0000,11728.0601
EC00529=0.0000,11731.4498
EC00530=0.0000,11734.1627
EC00531=0.0000,11735.7411
EC00532=0.0000,11735.9150
EC00533=0.0000,11735.8901
EC00534=0.0000,11735.8871
EC00535=0.0000,11736.1114
EC00536=0.0000,11737.1942
EC00537=0.0000,11740.0690
EC00538=0.0000,11742.7235
EC00539=0.0000,11745.0000
EC00540=0.0000,11747.2759
EC00541=0.0000,11749.9310
EC00542=0.0000,11752.8058
EC00543=0.0000,11753.8886
EC00544=0.0000,11754.1129
EC00545=0.0000,11754.1099
EC00546=0.0000,11754.0850
EC00547=0.0000,11754.2589
EC00548=0.0000,11755.8373
EC00549=0.0000,11758.5502
EC00550=0.0000,11761.9399
EC00551=0.0000,11765.6205
EC00552=0.0000,11769.3795
EC00553=0.0000,11773.0600
EC00554=0.0000,11776.4497
EC00555=0.0000,11779.1629
EC00556=0.0000,11780.7411
EC00557=0.0000,11780.9151
EC00558=0.0000,11780.8898
EC00559=0.0000,11780.8874
EC00560=0.0000,11781.1119
EC00561=0.0000,11782.1937
EC00562=0.0000,11785.0690
EC00563=0.0000,11787.7239
EC00564=0.0000,11790.0000
EC00565=0.0000,11790.0000
EC00566=0.0000,11792.2761
EC00567=0.0000,11794.9310
EC00568=0.0000,11797.8063
EC00569=0.0000,11798.8881
EC00570=0.0000,11799.1126
EC00571=0.0000,11799.1102
EC00572=0.0000,11799.0849
EC00573=0.0000,11799.2589
EC00574=0.0000,11800.8371
EC00575=0.0000,11803.5503
EC00576=0.0000,11806.9400
EC00577=0.0000,11810.6205
EC00578=0.0000,11814.3795
EC00579=0.0000,11818.0601
EC00580=0.0000,11821.4498
EC00581=0.0000,11824.1627
EC00582=0.0000,11825.7411
EC00583=0.0000,11825.9150
EC00584=0.0000,11825.8901
EC00585=0.0000,11825.8871
EC00586=0.0000,11826.1114
EC00587=0.0000,11827.1942
EC00588=0.0000,11830.0690
EC00589=0.0000,11832.7235
EC00590=0.0000,11835.0000
EC00591=0.0000,11837.2759
EC00592=0.0000,11839.9310
EC00593=0.0000,11842.8058
EC00594=0.0000,11843.8886
EC00595=0.0000,11844.1129
EC00596=0.0000,11844.1099
EC00597=0.0000,11844.0850
EC00598=0.0000,11844.2589
EC00599=0.0000,11845.8373
EC00600=0.0000,11848.5502
EC00601=0.0000,11851.9399
EC00602=0.0000,11855.6205
EC00603=0.0000,11859.3795
EC00604=0.0000,11863.0600
EC00605=0.0000,11866.4497
EC00606=0.0000,11869.1629
EC00607=0.0000,11870.7411
EC00608=0.0000,11870.9151
EC00609=0.0000,11870.8898
EC00610=0.0000,11870.8874
EC00611=0.0000,11871.1119
EC00612=0.0000,11872.1937
EC00613=0.0000,11875.0690
EC00614=0.0000,11877.7239
EC00615=0.0000,11880.0000
EC00616=0.0000,11882.2761
EC00617=0.0000,11884.9310
EC00618=0.0000,11887.8063
EC00619=0.0000,11888.8881
EC00620=0.0000,11889.1126
EC00621=0.0000,11889.1102
EC00622=0.0000,11889.0849
EC00623=0.0000,11889.2589
EC00624=0.0000,11890.8371
EC00625=0.0000,11893.5503
EC00626=0.0000,11896.9400
EC00627=0.0000,11900.6205
EC00628=0.0000,11904.3795
EC00629=0.0000,11908.0601
EC00630=0.0000,11911.4498
EC00631=0.0000,11914.1627
EC00632=0.0000,11915.7411
EC00633=0.0000,11915.9150
EC00634=0.0000,11915.8901
EC00635=0.0000,11915.8871
EC00636=0.0000,11916.1114
EC00637=0.0000,11917.1942
EC00638=0.0000,11920.0690
EC00639=0.0000,11922.7235
EC00640=0.0000,11925.0000
EC00641=0.0000,11927.2759
EC00642=0.0000,11929.9310
EC00643=0.0000,11932.8058
EC00644=0.0000,11933.8886
EC00645=0.0000,11934.1129
EC00646=0.0000,11934.1099
EC00647=0.0000,11934.0850
EC00648=0.0000,11934.2589
EC00649=0.0000,11935.8373
EC00650=0.0000,11938.5502
EC00651=0.0000,11941.9399
EC00652=0.0000,11945.6205
EC00653=0.0000,11949.3795
EC00654=0.0000,11953.0600
EC00655=0.0000,11956.4497
EC00656=0.0000,11959.1629
EC00657=0.0000,11960.7411
EC00658=0.0000,11960.9151
EC00659=0.0000,11960.8898
EC00660=0.0000,11960.8874
EC00661=0.0000,11961.1119
EC00662=0.0000,11962.1937
EC00663=0.0000,11965.0690
EC00664=0.0000,11967.7239
EC00665=0.0000,11970.0000
EC00666=0.0000,11970.0000
EC00667=0.0000,11972.2137
EC00668=0.0000,11974.8488
EC00669=0.0000,11977.7390
EC00670=0.0000,11978.7837
EC00671=0.0000,11978.9651
EC00672=0.0000,11978.9329
EC00673=0.0000,11978.8862
EC00674=0.0000,11979.0366
EC00675=0.0000,11980.6278
EC00676=0.0000,11983.3823
EC00677=0.0000,11986.8314
EC00678=0.0000,11990.5837
EC00679=0.0000,11994.4165
EC00680=0.0000,11998.1685
EC00681=0.0000,12001.6178
EC00682=0.0000,12004.3719
EC00683=0.0000,12005.9638
EC00684=0.0000,12006.1137
EC00685=0.0000,12006.0668
EC00686=0.0000,12006.0347
EC00687=0.0000,12006.2163
EC00688=0.0000,12007.2611
EC00689=0.0000,12010.1513
EC00690=0.0000,12012.7862
EC00691=0.0000,12015.0000
EC00692=0.0000,12017.2138
EC00693=0.0000,12019.8487
EC00694=0.0000,12022.7389
EC00695=0.0000,12023.7837
EC00696=0.0000,12023.9653
EC00697=0.0000,12023.9332
EC00698=0.0000,12023.8863
EC00699=0.0000,12024.0362
EC00700=0.0000,12025.6281
EC00701=0.0000,12028.3822
EC00702=0.0000,12031.8315
EC00703=0.0000,12035.5835
EC00704=0.0000,12039.4163
EC00705=0.0000,12043.1686
EC00706=0.0000,12046.6177
EC00707=0.0000,12049.3722
EC00708=0.0000,12050.9634
EC00709=0.0000,12051.1138
EC00710=0.0000,12051.0671
EC00711=0.0000,12051.0349
EC00712=0.0000,12051.2163
EC00713=0.0000,12052.2610
EC00714=0.0000,12055.1512
EC00715=0.0000,12057.7863
EC00716=0.0000,12060.0000
EC00717=0.0000,12062.2137
EC00718=0.0000,12064.8488
EC00719=0.0000,12067.7390
EC00720=0.0000,12068.7837
EC00721=0.0000,12068.9651
EC00722=0.0000,12068.9329
EC00723=0.0000,12068.8862
EC00724=0.0000,12069.0366
EC00725=0.0000,12070.6278
EC00726=0.0000,12073.3823
EC00727=0.0000,12076.8314
EC00728=0.0000,12080.5837
EC00729=0.0000,12084.4165
EC00730=0.0000,12088.1685
EC00731=0.0000,12091.6178
EC00732=0.0000,12094.3719
EC00733=0.0000,12095.9638
EC00734=0.0000,12096.1137
EC00735=0.0000,12096.0668
EC00736=0.0000,12096.0347
EC00737=0.0000,12096.2163
EC00738=0.0000,12097.2611
EC00739=0.0000,12100.1513
EC00740=0.0000,12102.7862
EC00741=0.0000,12105.0000
EC00742=0.0000,12107.2138
EC00743=0.0000,12109.8487
EC00744=0.0000,12112.7389
EC00745=0.0000,12113.7837
EC00746=0.0000,12113.9653
EC00747=0.0000,12113.9332
EC00748=0.0000,12113.8863
EC00749=0.0000,12114.0362
EC00750=0.0000,12115.6281
EC00751=0.0000,12118.3822
EC00752=0.0000,12121.8315
EC00753=0.0000,12125.5835
EC00754=0.0000,12129.4163
EC00755=0.0000,12133.1686
EC00756=0.0000,12136.6177
EC00757=0.0000,12139.3722
EC00758=0.0000,12140.9634
EC00759=0.0000,12141.1138
EC00760=0.0000,12141.0671
EC00761=0.0000,12141.0349
EC00762=0.0000,12141.2163
EC00763=0.0000,12142.2610
EC00764=0.0000,12145.1512
EC00765=0.0000,12147.7863
EC00766=0.0000,12150.0000
EC00767=0.0000,12150.0000
EC00768=0.0000,12152.2137
EC00769=0.0000,12154.8488
EC00770=0.0000,12157.7390
EC00771=0.0000,12158.7837
EC00772=0.0000,12158.9651
EC00773=0.0000,12158.9329
EC00774=0.0000,12158.8862
EC00775=0.0000,12159.0366
EC00776=0.0000,12160.6278
EC00777=0.0000,12163.3823
EC00778=0.0000,12166.8314
EC00779=0.0000,12170.5837
EC00780=0.0000,12174.4165
EC00781=0.0000,12178.1685
EC00782=0.0000,12181.6178
EC00783=0.0000,12184.3719
EC00784=0.0000,12185.9638
EC00785=0.0000,12186.1137
EC00786=0.0000,12186.0668
EC00787=0.0000,12186.0347
EC00788=0.0000,12186.2163
EC00789=0.0000,12187.2611
EC00790=0.0000,12190.1513
EC00791=0.0000,12192.7862
EC00792=0.0000,12195.0000
EC00793=0.0000,12197.2138
EC00794=0.0000,12199.8487
EC00795=0.0000,12202.7389
EC00796=0.0000,12203.7837
EC00797=0.0000,12203.9653
EC00798=0.0000,12203.9332
EC00799=0.0000,12203.8863
EC00800=0.0000,12204.0362
EC00801=0.0000,12205.6281
EC00802=0.0000,12208.3822
EC00803=0.0000,12211.8315
EC00804=0.0000,12215.5835
EC00805=0.0000,12219.4163
EC00806=0.0000,12223.1686
EC00807=0.0000,12226.6177
EC00808=0.0000,12229.3722
EC00809=0.0000,12230.9634
EC00810=0.0000,12231.1138
EC00811=0.0000,12231.0671
EC00812=0.0000,12231.0349
EC00813=0.0000,12231.2163
EC00814=0.0000,12232.2610
EC00815=0.0000,12235.1512
EC00816=0.0000,12237.7863
EC00817=0.0000,12240.0000
EC00818=0.0000,12242.2137
EC00819=0.0000,12244.8488
EC00820=0.0000,12247.7390
EC00821=0.0000,12248.7837
EC00822=0.0000,12248.9651
EC00823=0.0000,12248.9329
EC00824=0.0000,12248.8862
EC00825=0.0000,12249.0366
EC00826=0.0000,12250.6278
EC00827=0.0000,12253.3823
EC00828=0.0000,12256.8314
EC00829=0.0000,12260.5837
EC00830=0.0000,12264.4165
EC00831=0.0000,12268.1685
EC00832=0.0000,12271.6178
EC00833=0.0000,12274.3719
EC00834=0.0000,12275.9638
EC00835=0.0000,12276.1137
EC00836=0.0000,12276.0668
EC00837=0.0000,12276.0347
EC00838=0.0000,12276.2163
EC00839=0.0000,12277.2611
EC00840=0.0000,12280.1513
EC00841=0.0000,12282.7862
EC00842=0.0000,12285.0000
EC00843=0.0000,12287.2138
EC00844=0.0000,12289.8487
EC00845=0.0000,12292.7389
EC00846=0.0000,12293.7837
EC00847=0.0000,12293.9653
EC00848=0.0000,12293.9332
EC00849=0.0000,12293.8863
EC00850=0.0000,12294.0362
EC00851=0.0000,12295.6281
EC00852=0.0000,12298.3822
EC00853=0.0000,12301.8315
EC00854=0.0000,12305.5835
EC00855=0.0000,12309.4163
EC00856=0.0000,12313.1686
EC00857=0.0000,12316.6177
EC00858=0.0000,12319.3722
EC00859=0.0000,12320.9634
EC00860=0.0000,12321.1138
EC00861=0.0000,12321.0671
EC00862=0.0000,12321.0349
EC00863=0.0000,12321.2163
EC00864=0.0000,12322.2610
EC00865=0.0000,12325.1512
EC00866=0.0000,12327.7863
EC00867=0.0000,12330.0000
EC00868=0.0000,12330.0000
EC00869=0.0000,12332.1497
EC00870=0.0000,12334.7644
EC00871=0.0000,12337.6702
EC00872=0.0000,12338.6786
EC00873=0.0000,12338.8182
EC00874=0.0000,12338.7594
EC00875=0.0000,12338.6938
EC00876=0.0000,12338.8243
EC00877=0.0000,12340.4296
EC00878=0.0000,12343.2238
EC00879=0.0000,12346.7302
EC00880=0.0000,12350.5487
EC00881=0.0000,12354.4516
EC00882=0.0000,12358.2700
EC00883=0.0000,12361.7764
EC00884=0.0000,12364.5698
EC00885=0.0000,12366.1755
EC00886=0.0000,12366.3059
EC00887=0.0000,12366.2401
EC00888=0.0000,12366.1817
EC00889=0.0000,12366.3218
EC00890=0.0000,12367.3300
EC00891=0.0000,12370.2352
EC00892=0.0000,12372.8504
EC00893=0.0000,12375.0000
EC00894=0.0000,12377.1496
EC00895=0.0000,12379.7648
EC00896=0.0000,12382.6700
EC00897=0.0000,12383.6782
EC00898=0.0000,12383.8183
EC00899=0.0000,12383.7599
EC00900=0.0000,12383.6941
EC00901=0.0000,12383.8245
EC00902=0.0000,12385.4302
EC00903=0.0000,12388.2236
EC00904=0.0000,12391.7300
EC00905=0.0000,12395.5484
EC00906=0.0000,12399.4513
EC00907=0.0000,12403.2698
EC00908=0.0000,12406.7762
EC00909=0.0000,12409.5704
EC00910=0.0000,12411.1757
EC00911=0.0000,12411.3062
EC00912=0.0000,12411.2406
EC00913=0.0000,12411.1818
EC00914=0.0000,12411.3214
EC00915=0.0000,12412.3298
EC00916=0.0000,12415.2356
EC00917=0.0000,12417.8503
EC00918=0.0000,12420.0000
EC00919=0.0000,12422.1497
EC00920=0.0000,12424.7644
EC00921=0.0000,12427.6701
EC00922=0.0000,12428.6786
EC00923=0.0000,12428.8182
EC00924=0.0000,12428.7594
EC00925=0.0000,12428.6938
EC00926=0.0000,12428.8243
EC00927=0.0000,12430.4296
EC00928=0.0000,12433.2238
EC00929=0.0000,12436.7302
EC00930=0.0000,12440.5487
EC00931=0.0000,12444.4516
EC00932=0.0000,12448.2700
EC00933=0.0000,12451.7764
EC00934=0.0000,12454.5698
EC00935=0.0000,12456.1755
EC00936=0.0000,12456.3059
EC00937=0.0000,12456.2401
EC00938=0.0000,12456.1817
EC00939=0.0000,12456.3218
EC00940=0.0000,12457.3300
EC00941=0.0000,12460.2352
EC00942=0.0000,12462.8504
EC00943=0.0000,12465.0000
EC00944=0.0000,12467.1496
EC00945=0.0000,12469.7648
EC00946=0.0000,12472.6700
EC00947=0.0000,12473.6782
EC00948=0.0000,12473.8183
EC00949=0.0000,12473.7599
EC00950=0.0000,12473.6941
EC00951=0.0000,12473.8245
EC00952=0.0000,12475.4302
EC00953=0.0000,12478.2236
EC00954=0.0000,12481.7300
EC00955=0.0000,12485.5484
EC00956=0.0000,12489.4513
EC00957=0.0000,12493.2698
EC00958=0.0000,12496.7762
EC00959=0.0000,12499.5704
EC00960=0.0000,12501.1757
EC00961=0.0000,12501.3062
EC00962=0.0000,12501.2406
EC00963=0.0000,12501.1818
EC00964=0.0000,12501.3214
EC00965=0.0000,12502.3298
EC00966=0.0000,12505.2356
EC00967=0.0000,12507.8503
EC00968=0.0000,12510.0000
EC00969=0.0000,12510.0000
EC00970=0.0000,12512.1497
EC00971=0.0000,12514.7644
EC00972=0.0000,12517.6701
EC00973=0.0000,12518.6786
EC00974=0.0000,12518.8182
EC00975=0.0000,12518.7594
EC00976=0.0000,12518.6938
EC00977=0.0000,12518.8243
EC00978=0.0000,12520.4296
EC00979=0.0000,12523.2238
EC00980=0.0000,12526.7302
EC00981=0.0000,12530.5487
EC00982=0.0000,12534.4516
EC00983=0.0000,12538.2700
EC00984=0.0000,12541.7764
EC00985=0.0000,12544.5698
EC00986=0.0000,12546.1755
EC00987=0.0000,12546.3059
EC00988=0.0000,12546.2401
EC00989=0.0000,12546.1817
EC00990=0.0000,12546.3218
EC00991=0.0000,12547.3300
EC00992=0.0000,12550.2352
EC00993=0.0000,12552.8504
EC00994=0.0000,12555.0000
EC00995=0.0000,12557.1496
EC00996=0.0000,12559.7648
EC00997=0.0000,12562.6700
EC00998=0.0000,12563.6782
EC00999=0.0000,12563.8183
EC01000=0.0000,12563.7599
EC01001=0.0000,12563.6941
EC01002=0.0000,12563.8245
EC01003=0.0000,12565.4302
EC01004=0.0000,12568.2236
EC01005=0.0000,12571.7300
EC01006=0.0000,12575.5484
EC01007=0.0000,12579.4513
EC01008=0.0000,12583.2698
EC01009=0.0000,12586.7762
EC01010=0.0000,12589.5704
EC01011=0.0000,12591.1757
EC01012=0.0000,12591.3062
EC01013=0.0000,12591.2406
EC01014=0.0000,12591.1818
EC01015=0.0000,12591.3214
EC01016=0.0000,12592.3298
EC01017=0.0000,12595.2356
EC01018=0.0000,12597.8503
EC01019=0.0000,12600.0000
EC01020=0.0000,12602.1497
EC01021=0.0000,12604.7644
EC01022=0.0000,12607.6701
EC01023=0.0000,12608.6786
EC01024=0.0000,12608.8182
EC01025=0.0000,12608.7594
EC01026=0.0000,12608.6938
EC01027=0.0000,12608.8243
EC01028=0.0000,12610.4296
EC01029=0.0000,12613.2238
EC01030=0.0000,12616.7302
EC01031=0.0000,12620.5487
EC01032=0.0000,12624.4516
EC01033=0.0000,12628.2700
EC01034=0.0000,12631.7764
EC01035=0.0000,12634.5698
EC01036=0.0000,12636.1755
EC01037=0.0000,12636.3059
EC01038=0.0000,12636.2401
EC01039=0.0000,12636.1817
EC01040=0.0000,12636.3218
EC01041=0.0000,12637.3300
EC01042=0.0000,12640.2352
EC01043=0.0000,12642.8504
EC01044=0.0000,12645.0000
EC01045=0.0000,12647.1496
EC01046=0.0000,12649.7648
EC01047=0.0000,12652.6700
EC01048=0.0000,12653.6782
EC01049=0.0000,12653.8183
EC01050=0.0000,12653.7599
EC01051=0.0000,12653.6941
EC01052=0.0000,12653.8245
EC01053=0.0000,12655.4302
EC01054=0.0000,12658.2236
EC01055=0.0000,12661.7300
EC01056=0.0000,12665.5484
EC01057=0.0000,12669.4513
EC01058=0.0000,12673.2698
EC01059=0.0000,12676.7762
EC01060=0.0000,12679.5704
EC01061=0.0000,12681.1757
EC01062=0.0000,12681.3062
EC01063=0.0000,12681.2406
EC01064=0.0000,12681.1818
EC01065=0.0000,12681.3214
EC01066=0.0000,12682.3299
EC01067=0.0000,12685.2356
EC01068=0.0000,12687.8503
EC01069=0.0000,12690.0000
EC01070=0.0000,12690.0000
EC01071=0.0000,12692.0841
EC01072=0.0000,12694.6784
EC01073=0.0000,12697.6002
EC01074=0.0000,12698.5715
EC01075=0.0000,12698.6723
EC01076=0.0000,12698.5913
EC01077=0.0000,12698.5111
EC01078=0.0000,12698.6248
EC01079=0.0000,12700.2442
EC01080=0.0000,12703.0758
EC01081=0.0000,12706.6354
EC01082=0.0000,12710.5162
EC01083=0.0000,12714.4836
EC01084=0.0000,12718.3648
EC01085=0.0000,12721.9242
EC01086=0.0000,12724.7559
EC01087=0.0000,12726.3755
EC01088=0.0000,12726.4893
EC01089=0.0000,12726.4090
EC01090=0.0000,12726.3280
EC01091=0.0000,12726.4285
EC01092=0.0000,12727.4001
EC01093=0.0000,12730.3225
EC01094=0.0000,12732.9160
EC01095=0.0000,12735.0000
EC01096=0.0000,12737.0840
EC01097=0.0000,12739.6788
EC01098=0.0000,12742.5999
EC01099=0.0000,12743.5715
EC01100=0.0000,12743.6720
EC01101=0.0000,12743.5910
EC01102=0.0000,12743.5107
EC01103=0.0000,12743.6245
EC01104=0.0000,12745.2441
EC01105=0.0000,12748.0758
EC01106=0.0000,12751.6352
EC01107=0.0000,12755.5164
EC01108=0.0000,12759.4838
EC01109=0.0000,12763.3646
EC01110=0.0000,12766.9242
EC01111=0.0000,12769.7558
EC01112=0.0000,12771.3752
EC01113=0.0000,12771.4889
EC01114=0.0000,12771.4087
EC01115=0.0000,12771.3277
EC01116=0.0000,12771.4285
EC01117=0.0000,12772.3998
EC01118=0.0000,12775.3216
EC01119=0.0000,12777.9159
EC01120=0.0000,12780.0000
EC01121=0.0000,12782.0841
EC01122=0.0000,12784.6784
EC01123=0.0000,12787.6002
EC01124=0.0000,12788.5715
EC01125=0.0000,12788.6723
EC01126=0.0000,12788.5913
EC01127=0.0000,12788.5111
EC01128=0.0000,12788.6248
EC01129=0.0000,12790.2442
EC01130=0.0000,12793.0758
EC01131=0.0000,12796.6354
EC01132=0.0000,12800.5162
EC01133=0.0000,12804.4836
EC01134=0.0000,12808.3648
EC01135=0.0000,12811.9242
EC01136=0.0000,12814.7559
EC01137=0.0000,12816.3755
EC01138=0.0000,12816.4893
EC01139=0.0000,12816.4090
EC01140=0.0000,12816.3280
EC01141=0.0000,12816.4285
EC01142=0.0000,12817.4001
EC01143=0.0000,12820.3225
EC01144=0.0000,12822.9160
EC01145=0.0000,12825.0000
EC01146=0.0000,12827.0840
EC01147=0.0000,12829.6788
EC01148=0.0000,12832.5999
EC01149=0.0000,12833.5715
EC01150=0.0000,12833.6720
EC01151=0.0000,12833.5910
EC01152=0.0000,12833.5107
EC01153=0.0000,12833.6245
EC01154=0.0000,12835.2441
EC01155=0.0000,12838.0758
EC01156=0.0000,12841.6352
EC01157=0.0000,12845.5164
EC01158=0.0000,12849.4838
EC01159=0.0000,12853.3646
EC01160=0.0000,12856.9242
EC01161=0.0000,12859.7558
EC01162=0.0000,12861.3752
EC01163=0.0000,12861.4889
EC01164=0.0000,12861.4087
EC01165=0.0000,12861.3277
EC01166=0.0000,12861.4285
EC01167=0.0000,12862.3998
EC01168=0.0000,12865.3216
EC01169=0.0000,12867.9159
EC01170=0.0000,12870.0000
EC01171=0.0000,12870.0000
EC01172=0.0000,12872.0841
EC01173=0.0000,12874.6784
EC01174=0.0000,12877.6002
EC01175=0.0000,12878.5715
EC01176=0.0000,12878.6723
EC01177=0.0000,12878.5913
EC01178=0.0000,12878.5111
EC01179=0.0000,12878.6248
EC01180=0.0000,12880.2442
EC01181=0.0000,12883.0758
EC01182=0.0000,12886.6354
EC01183=0.0000,12890.5162
EC01184=0.0000,12894.4836
EC01185=0.0000,12898.3648
EC01186=0.0000,12901.9242
EC01187=0.0000,12904.7559
EC01188=0.0000,12906.3755
EC01189=0.0000,12906.4893
EC01190=0.0000,12906.4090
EC01191=0.0000,12906.3280
EC01192=0.0000,12906.4285
EC01193=0.0000,12907.4001
EC01194=0.0000,12910.3225
EC01195=0.0000,12912.9160
EC01196=0.0000,12915.0000
EC01197=0.0000,12917.0840
EC01198=0.0000,12919.6788
EC01199=0.0000,12922.5999
EC01200=0.0000,12923.5715
EC01201=0.0000,12923.6720
EC01202=0.0000,12923.5910
EC01203=0.0000,12923.5107
EC01204=0.0000,12923.6245
EC01205=0.0000,12925.2441
EC01206=0.0000,12928.0758
EC01207=0.0000,12931.6352
EC01208=0.0000,12935.5164
EC01209=0.0000,12939.4838
EC01210=0.0000,12943.3646
EC01211=0.0000,12946.9242
EC01212=0.0000,12949.7558
EC01213=0.0000,12951.3752
EC01214=0.0000,12951.4889
EC01215=0.0000,12951.4087
EC01216=0.0000,12951.3277
EC01217=0.0000,12951.4285
EC01218=0.0000,12952.3998
EC01219=0.0000,12955.3216
EC01220=0.0000,12957.9159
EC01221=0.0000,12960.0000
EC01222=0.0000,12962.0841
EC01223=0.0000,12964.6784
EC01224=0.0000,12967.6002
EC01225=0.0000,12968.5715
EC01226=0.0000,12968.6723
EC01227=0.0000,12968.5913
EC01228=0.0000,12968.5111
EC01229=0.0000,12968.6248
EC01230=0.0000,12970.2442
EC01231=0.0000,12973.0758
EC01232=0.0000,12976.6354
EC01233=0.0000,12980.5162
EC01234=0.0000,12984.4836
EC01235=0.0000,12988.3648
EC01236=0.0000,12991.9242
EC01237=0.0000,12994.7559
EC01238=0.0000,12996.3755
EC01239=0.0000,12996.4893
EC01240=0.0000,12996.4090
EC01241=0.0000,12996.3280
EC01242=0.0000,12996.4285
EC01243=0.0000,12997.4001
EC01244=0.0000,13000.3225
EC01245=0.0000,13002.9160
EC01246=0.0000,13005.0000
EC01247=0.0000,13007.0840
EC01248=0.0000,13009.6788
EC01249=0.0000,13012.5999
EC01250=0.0000,13013.5715
EC01251=0.0000,13013.6720
EC01252=0.0000,13013.5910
EC01253=0.0000,13013.5107
EC01254=0.0000,13013.6245
EC01255=0.0000,13015.2441
EC01256=0.0000,13018.0758
EC01257=0.0000,13021.6352
EC01258=0.0000,13025.5164
EC01259=0.0000,13029.4838
EC01260=0.0000,13033.3646
EC01261=0.0000,13036.9242
EC01262=0.0000,13039.7558
EC01263=0.0000,13041.3752
EC01264=0.0000,13041.4889
EC01265=0.0000,13041.4087
EC01266=0.0000,13041.3277
EC01267=0.0000,13041.4285
EC01268=0.0000,13042.3998
EC01269=0.0000,13045.3216
EC01270=0.0000,13047.9159
EC01271=0.0000,13050.0000
EC01272=0.0000,13050.0000
EC01273=0.0000,13052.0177
EC01274=0.0000,13054.5896
EC01275=0.0000,13057.5288
EC01276=0.0000,13058.4644
EC01277=0.0000,13058.5281
EC01278=0.0000,13058.4283
EC01279=0.0000,13058.3383
EC01280=0.0000,13058.4379
EC01281=0.0000,13060.0717
EC01282=0.0000,13062.9390
EC01283=0.0000,13066.5485
EC01284=0.0000,13070.4866
EC01285=0.0000,13074.5131
EC01286=0.0000,13078.4517
EC01287=0.0000,13082.0609
EC01288=0.0000,13084.9281
EC01289=0.0000,13086.5622
EC01290=0.0000,13086.6621
EC01291=0.0000,13086.5714
EC01292=0.0000,13086.4714
EC01293=0.0000,13086.5356
EC01294=0.0000,13087.4711
EC01295=0.0000,13090.4108
EC01296=0.0000,13092.9827
EC01297=0.0000,13095.0000
EC01298=0.0000,13097.0166
EC01299=0.0000,13099.5906
EC01300=0.0000,13102.5289
EC01301=0.0000,13103.4644
EC01302=0.0000,13103.5286
EC01303=0.0000,13103.4286
EC01304=0.0000,13103.3379
EC01305=0.0000,13103.4378
EC01306=0.0000,13105.0719
EC01307=0.0000,13107.9391
EC01308=0.0000,13111.5483
EC01309=0.0000,13115.4869
EC01310=0.0000,13119.5134
EC01311=0.0000,13123.4515
EC01312=0.0000,13127.0610
EC01313=0.0000,13129.9283
EC01314=0.0000,13131.5621
EC01315=0.0000,13131.6617
EC01316=0.0000,13131.5717
EC01317=0.0000,13131.4719
EC01318=0.0000,13131.5356
EC01319=0.0000,13132.4712
EC01320=0.0000,13135.4104
EC01321=0.0000,13137.9823
EC01322=0.0000,13140.0000
EC01323=0.0000,13142.0167
EC01324=0.0000,13144.5896
EC01325=0.0000,13147.5286
EC01326=0.0000,13148.4644
EC01327=0.0000,13148.5281
EC01328=0.0000,13148.4283
EC01329=0.0000,13148.3383
EC01330=0.0000,13148.4379
EC01331=0.0000,13150.0717
EC01332=0.0000,13152.9390
EC01333=0.0000,13156.5485
EC01334=0.0000,13160.4866
EC01335=0.0000,13164.5131
EC01336=0.0000,13168.4517
EC01337=0.0000,13172.0609
EC01338=0.0000,13174.9281
EC01339=0.0000,13176.5622
EC01340=0.0000,13176.6621
EC01341=0.0000,13176.5714
EC01342=0.0000,13176.4714
EC01343=0.0000,13176.5356
EC01344=0.0000,13177.4711
EC01345=0.0000,13180.4108
EC01346=0.0000,13182.9827
EC01347=0.0000,13185.0000
EC01348=0.0000,13187.0166
EC01349=0.0000,13189.5906
EC01350=0.0000,13192.5289
EC01351=0.0000,13193.4644
EC01352=0.0000,13193.5286
EC01353=0.0000,13193.4286
EC01354=0.0000,13193.3379
EC01355=0.0000,13193.4378
EC01356=0.0000,13195.0719
EC01357=0.0000,13197.9391
EC01358=0.0000,13201.5483
EC01359=0.0000,13205.4869
EC01360=0.0000,13209.5134
EC01361=0.0000,13213.4515
EC01362=0.0000,13217.0610
EC01363=0.0000,13219.9283
EC01364=0.0000,13221.5621
EC01365=0.0000,13221.6617
EC01366=0.0000,13221.5717
EC01367=0.0000,13221.4719
EC01368=0.0000,13221.5356
EC01369=0.0000,13222.4712
EC01370=0.0000,13225.4104
EC01371=0.0000,13227.9823
EC01372=0.0000,13230.0000
EC01373=0.0000,13230.0000
EC01374=0.0000,13232.0167
EC01375=0.0000,13234.5896
EC01376=0.0000,13237.5286
EC01377=0.0000,13238.4644
EC01378=0.0000,13238.5281
EC01379=0.0000,13238.4283
EC01380=0.0000,13238.3383
EC01381=0.0000,13238.4379
EC01382=0.0000,13240.0717
EC01383=0.0000,13242.9390
EC01384=0.0000,13246.5485
EC01385=0.0000,13250.4866
EC01386=0.0000,13254.5131
EC01387=0.0000,13258.4517
EC01388=0.0000,13262.0609
EC01389=0.0000,13264.9281
EC01390=0.0000,13266.5622
EC01391=0.0000,13266.6621
EC01392=0.0000,13266.5714
EC01393=0.0000,13266.4714
EC01394=0.0000,13266.5356
EC01395=0.0000,13267.4711
EC01396=0.0000,13270.4108
EC01397=0.0000,13272.9827
EC01398=0.0000,13275.0000
EC01399=0.0000,13277.0166
EC01400=0.0000,13279.5906
EC01401=0.0000,13282.5289
EC01402=0.0000,13283.4644
EC01403=0.0000,13283.5286
EC01404=0.0000,13283.4286
EC01405=0.0000,13283.3379
EC01406=0.0000,13283.4378
EC01407=0.0000,13285.0719
EC01408=0.0000,13287.9391
EC01409=0.0000,13291.5483
EC01410=0.0000,13295.4869
EC01411=0.0000,13299.5134
EC01412=0.0000,13303.4515
EC01413=0.0000,13307.0610
EC01414=0.0000,13309.9283
EC01415=0.0000,13311.5621
EC01416=0.0000,13311.6617
EC01417=0.0000,13311.5717
EC01418=0.0000,13311.4719
EC01419=0.0000,13311.5356
EC01420=0.0000,13312.4712
EC01421=0.0000,13315.4104
EC01422=0.0000,13317.9823
EC01423=0.0000,13320.0000
EC01424=0.0000,13322.0167
EC01425=0.0000,13324.5896
EC01426=0.0000,13327.5286
EC01427=0.0000,13328.4644
EC01428=0.0000,13328.5281
EC01429=0.0000,13328.4283
EC01430=0.0000,13328.3383
EC01431=0.0000,13328.4379
EC01432=0.0000,13330.0717
EC01433=0.0000,13332.9390
EC01434=0.0000,13336.5485
EC01435=0.0000,13340.4866
EC01436=0.0000,13344.5131
EC01437=0.0000,13348.4517
EC01438=0.0000,13352.0609
EC01439=0.0000,13354.9281
EC01440=0.0000,13356.5622
EC01441=0.0000,13356.6621
EC01442=0.0000,13356.5714
EC01443=0.0000,13356.4714
EC01444=0.0000,13356.5356
EC01445=0.0000,13357.4711
EC01446=0.0000,13360.4108
EC01447=0.0000,13362.9827
EC01448=0.0000,13365.0000
EC01449=0.0000,13367.0166
EC01450=0.0000,13369.5906
EC01451=0.0000,13372.5289
EC01452=0.0000,13373.4644
EC01453=0.0000,13373.5286
EC01454=0.0000,13373.4286
EC01455=0.0000,13373.3379
EC01456=0.0000,13373.4378
EC01457=0.0000,13375.0719
EC01458=0.0000,13377.9391
EC01459=0.0000,13381.5483
EC01460=0.0000,13385.4869
EC01461=0.0000,13389.5134
EC01462=0.0000,13393.4515
EC01463=0.0000,13397.0610
EC01464=0.0000,13399.9283
EC01465=0.0000,13401.5621
EC01466=0.0000,13401.6617
EC01467=0.0000,13401.5717
EC01468=0.0000,13401.4719
EC01469=0.0000,13401.5356
EC01470=0.0000,13402.4714
EC01471=0.0000,13405.4104
EC01472=0.0000,13407.9833
EC01473=0.0000,13410.0000
EC01474=0.0000,13410.0000
EC01475=0.0000,13411.9494
EC01476=0.0000,13414.4996
EC01477=0.0000,13417.4570
EC01478=0.0000,13418.3570
EC01479=0.0000,13418.3879
EC01480=0.0000,13418.2735
EC01481=0.0000,13418.1767
EC01482=0.0000,13418.2659
EC01483=0.0000,13419.9145
EC01484=0.0000,13422.8156
EC01485=0.0000,13426.4700
EC01486=0.0000,13430.4601
EC01487=0.0000,13434.5401
EC01488=0.0000,13438.5303
EC01489=0.0000,13442.1847
EC01490=0.0000,13445.0854
EC01491=0.0000,13446.7338
EC01492=0.0000,13446.8229
EC01493=0.0000,13446.7263
EC01494=0.0000,13446.6122
EC01495=0.0000,13446.6435
EC01496=0.0000,13447.5429
EC01497=0.0000,13450.5003
EC01498=0.0000,13453.0512
EC01499=0.0000,13455.0000
EC01500=0.0000,13456.9488
EC01501=0.0000,13459.5003
EC01502=0.0000,13462.4571
EC01503=0.0000,13463.3565
EC01504=0.0000,13463.3878
EC01505=0.0000,13463.2737
EC01506=0.0000,13463.1771
EC01507=0.0000,13463.2662
EC01508=0.0000,13464.9146
EC01509=0.0000,13467.8153
EC01510=0.0000,13471.4697
EC01511=0.0000,13475.4599
EC01512=0.0000,13479.5399
EC01513=0.0000,13483.5300
EC01514=0.0000,13487.1844
EC01515=0.0000,13490.0855
EC01516=0.0000,13491.7341
EC01517=0.0000,13491.8233
EC01518=0.0000,13491.7265
EC01519=0.0000,13491.6121
EC01520=0.0000,13491.6430
EC01521=0.0000,13492.5430
EC01522=0.0000,13495.5004
EC01523=0.0000,13498.0506
EC01524=0.0000,13500.0000
EC01525=0.0000,13501.9484
EC01526=0.0000,13504.5006
EC01527=0.0000,13507.4570
EC01528=0.0000,13508.3570
EC01529=0.0000,13508.3879
EC01530=0.0000,13508.2735
EC01531=0.0000,13508.1767
EC01532=0.0000,13508.2659
EC01533=0.0000,13509.9145
EC01534=0.0000,13512.8156
EC01535=0.0000,13516.4700
EC01536=0.0000,13520.4601
EC01537=0.0000,13524.5401
EC01538=0.0000,13528.5303
EC01539=0.0000,13532.1847
EC01540=0.0000,13535.0854
EC01541=0.0000,13536.7338
EC01542=0.0000,13536.8229
EC01543=0.0000,13536.7263
EC01544=0.0000,13536.6122
EC01545=0.0000,13536.6435
EC01546=0.0000,13537.5429
EC01547=0.0000,13540.5003
EC01548=0.0000,13543.0512
EC01549=0.0000,13545.0000
EC01550=0.0000,13546.9488
EC01551=0.0000,13549.5003
EC01552=0.0000,13552.4571
EC01553=0.0000,13553.3565
EC01554=0.0000,13553.3878
EC01555=0.0000,13553.2737
EC01556=0.0000,13553.1771
EC01557=0.0000,13553.2662
EC01558=0.0000,13554.9146
EC01559=0.0000,13557.8153
EC01560=0.0000,13561.4697
EC01561=0.0000,13565.4599
EC01562=0.0000,13569.5399
EC01563=0.0000,13573.5300
EC01564=0.0000,13577.1844
EC01565=0.0000,13580.0855
EC01566=0.0000,13581.7341
EC01567=0.0000,13581.8233
EC01568=0.0000,13581.7265
EC01569=0.0000,13581.6121
EC01570=0.0000,13581.6430
EC01571=0.0000,13582.5430
EC01572=0.0000,13585.5004
EC01573=0.0000,13588.0506
EC01574=0.0000,13590.0000
EC01575=0.0000,13590.0000
EC01576=0.0000,13591.9484
EC01577=0.0000,13594.5006
EC01578=0.0000,13597.4570
EC01579=0.0000,13598.3570
EC01580=0.0000,13598.3879
EC01581=0.0000,13598.2735
EC01582=0.0000,13598.1767
EC01583=0.0000,13598.2659
EC01584=0.0000,13599.9145
EC01585=0.0000,13602.8156
EC01586=0.0000,13606.4700
EC01587=0.0000,13610.4601
EC01588=0.0000,13614.5401
EC01589=0.0000,13618.5303
EC01590=0.0000,13622.1847
EC01591=0.0000,13625.0854
EC01592=0.0000,13626.7338
EC01593=0.0000,13626.8229
EC01594=0.0000,13626.7263
EC01595=0.0000,13626.6122
EC01596=0.0000,13626.6435
EC01597=0.0000,13627.5429
EC01598=0.0000,13630.5003
EC01599=0.0000,13633.0512
EC01600=0.0000,13635.0000
EC01601=0.0000,13636.9488
EC01602=0.0000,13639.5003
EC01603=0.0000,13642.4571
EC01604=0.0000,13643.3565
EC01605=0.0000,13643.3878
EC01606=0.0000,13643.2737
EC01607=0.0000,13643.1771
EC01608=0.0000,13643.2662
EC01609=0.0000,13644.9146
EC01610=0.0000,13647.8153
EC01611=0.0000,13651.4697
EC01612=0.0000,13655.4599
EC01613=0.0000,13659.5399
EC01614=0.0000,13663.5300
EC01615=0.0000,13667.1844
EC01616=0.0000,13670.0855
EC01617=0.0000,13671.7341
EC01618=0.0000,13671.8233
EC01619=0.0000,13671.7265
EC01620=0.0000,13671.6121
EC01621=0.0000,13671.6430
EC01622=0.0000,13672.5430
EC01623=0.0000,13675.5004
EC01624=0.0000,13678.0506
EC01625=0.0000,13680.0000
EC01626=0.0000,13681.9484
EC01627=0.0000,13684.5006
EC01628=0.0000,13687.4570
EC01629=0.0000,13688.3570
EC01630=0.0000,13688.3879
EC01631=0.0000,13688.2735
EC01632=0.0000,13688.1767
EC01633=0.0000,13688.2659
EC01634=0.0000,13689.9145
EC01635=0.0000,13692.8156
EC01636=0.0000,13696.4700
EC01637=0.0000,13700.4601
EC01638=0.0000,13704.5401
EC01639=0.0000,13708.5303
EC01640=0.0000,13712.1847
EC01641=0.0000,13715.0854
EC01642=0.0000,13716.7338
EC01643=0.0000,13716.8229
EC01644=0.0000,13716.7263
EC01645=0.0000,13716.6122
EC01646=0.0000,13716.6435
EC01647=0.0000,13717.5429
EC01648=0.0000,13720.5003
EC01649=0.0000,13723.0512
EC01650=0.0000,13725.0000
EC01651=0.0000,13726.9488
EC01652=0.0000,13729.5003
EC01653=0.0000,13732.4571
EC01654=0.0000,13733.3565
EC01655=0.0000,13733.3878
EC01656=0.0000,13733.2737
EC01657=0.0000,13733.1771
EC01658=0.0000,13733.2662
EC01659=0.0000,13734.9146
EC01660=0.0000,13737.8153
EC01661=0.0000,13741.4697
EC01662=0.0000,13745.4599
EC01663=0.0000,13749.5399
EC01664=0.0000,13753.5300
EC01665=0.0000,13757.1844
EC01666=0.0000,13760.0855
EC01667=0.0000,13761.7341
EC01668=0.0000,13761.8233
EC01669=0.0000,13761.7265
EC01670=0.0000,13761.6121
EC01671=0.0000,13761.6430
EC01672=0.0000,13762.5430
EC01673=0.0000,13765.4994
EC01674=0.0000,13768.0516
EC01675=0.0000,13770.0000
EC01676=0.0000,13770.0000
EC01677=0.0000,13771.8799
EC01678=0.0000,13774.4091
EC01679=0.0000,13777.3837
EC01680=0.0000,13778.2508
EC01681=0.0000,13778.2514
EC01682=0.0000,13778.1286
EC01683=0.0000,13778.0287
EC01684=0.0000,13778.1105
EC01685=0.0000,13779.7738
EC01686=0.0000,13782.7052
EC01687=0.0000,13786.4001
EC01688=0.0000,13790.4362
EC01689=0.0000,13794.5637
EC01690=0.0000,13798.5997
EC01691=0.0000,13802.2952
EC01692=0.0000,13805.2262
EC01693=0.0000,13806.8889
EC01694=0.0000,13806.9711
EC01695=0.0000,13806.8716
EC01696=0.0000,13806.7487
EC01697=0.0000,13806.7500
EC01698=0.0000,13807.6160
EC01699=0.0000,13810.5914
EC01700=0.0000,13813.1202
EC01701=0.0000,13815.0000
EC01702=0.0000,13816.8791
EC01703=0.0000,13819.4092
EC01704=0.0000,13822.3840
EC01705=0.0000,13823.2500
EC01706=0.0000,13823.2513
EC01707=0.0000,13823.1284
EC01708=0.0000,13823.0289
EC01709=0.0000,13823.1111
EC01710=0.0000,13824.7738
EC01711=0.0000,13827.7048
EC01712=0.0000,13831.4003
EC01713=0.0000,13835.4363
EC01714=0.0000,13839.5638
EC01715=0.0000,13843.5999
EC01716=0.0000,13847.2948
EC01717=0.0000,13850.2262
EC01718=0.0000,13851.8895
EC01719=0.0000,13851.9713
EC01720=0.0000,13851.8714
EC01721=0.0000,13851.7486
EC01722=0.0000,13851.7492
EC01723=0.0000,13852.6163
EC01724=0.0000,13855.5909
EC01725=0.0000,13858.1201
EC01726=0.0000,13860.0000
EC01727=0.0000,13861.8799
EC01728=0.0000,13864.4091
EC01729=0.0000,13867.3837
EC01730=0.0000,13868.2508
EC01731=0.0000,13868.2514
EC01732=0.0000,13868.1286
EC01733=0.0000,13868.0287
EC01734=0.0000,13868.1105
EC01735=0.0000,13869.7738
EC01736=0.0000,13872.7052
EC01737=0.0000,13876.4001
EC01738=0.0000,13880.4362
EC01739=0.0000,13884.5637
EC01740=0.0000,13888.5997
EC01741=0.0000,13892.2952
EC01742=0.0000,13895.2262
EC01743=0.0000,13896.8889
EC01744=0.0000,13896.9711
EC01745=0.0000,13896.8716
EC01746=0.0000,13896.7487
EC01747=0.0000,13896.7500
EC01748=0.0000,13897.6160
EC01749=0.0000,13900.5914
EC01750=0.0000,13903.1202
EC01751=0.0000,13905.0000
EC01752=0.0000,13906.8791
EC01753=0.0000,13909.4092
EC01754=0.0000,13912.3840
EC01755=0.0000,13913.2500
EC01756=0.0000,13913.2513
EC01757=0.0000,13913.1284
EC01758=0.0000,13913.0289
EC01759=0.0000,13913.1111
EC01760=0.0000,13914.7738
EC01761=0.0000,13917.7048
EC01762=0.0000,13921.4003
EC01763=0.0000,13925.4363
EC01764=0.0000,13929.5638
EC01765=0.0000,13933.5999
EC01766=0.0000,13937.2948
EC01767=0.0000,13940.2262
EC01768=0.0000,13941.8895
EC01769=0.0000,13941.9713
EC01770=0.0000,13941.8714
EC01771=0.0000,13941.7486
EC01772=0.0000,13941.7492
EC01773=0.0000,13942.6163
EC01774=0.0000,13945.5909
EC01775=0.0000,13948.1201
EC01776=0.0000,13950.0000
EC01777=0.0000,13950.0000
EC01778=0.0000,13951.8799
EC01779=0.0000,13954.4091
EC01780=0.0000,13957.3837
EC01781=0.0000,13958.2508
EC01782=0.0000,13958.2514
EC01783=0.0000,13958.1286
EC01784=0.0000,13958.0287
EC01785=0.0000,13958.1105
EC01786=0.0000,13959.7738
EC01787=0.0000,13962.7052
EC01788=0.0000,13966.4001
EC01789=0.0000,13970.4362
EC01790=0.0000,13974.5637
EC01791=0.0000,13978.5997
EC01792=0.0000,13982.2952
EC01793=0.0000,13985.2262
EC01794=0.0000,13986.8889
EC01795=0.0000,13986.9711
EC01796=0.0000,13986.8716
EC01797=0.0000,13986.7487
EC01798=0.0000,13986.7500
EC01799=0.0000,13987.6160
EC01800=0.0000,13990.5914
EC01801=0.0000,13993.1202
EC01802=0.0000,13995.0000
EC01803=0.0000,13996.8791
EC01804=0.0000,13999.4092
EC01805=0.0000,14002.3840
EC01806=0.0000,14003.2500
EC01807=0.0000,14003.2513
EC01808=0.0000,14003.1284
EC01809=0.0000,14003.0289
EC01810=0.0000,14003.1111
EC01811=0.0000,14004.7738
EC01812=0.0000,14007.7048
EC01813=0.0000,14011.4003
EC01814=0.0000,14015.4363
EC01815=0.0000,14019.5638
EC01816=0.0000,14023.5999
EC01817=0.0000,14027.2948
EC01818=0.0000,14030.2262
EC01819=0.0000,14031.8895
EC01820=0.0000,14031.9713
EC01821=0.0000,14031.8714
EC01822=0.0000,14031.7486
EC01823=0.0000,14031.7492
EC01824=0.0000,14032.6163
EC01825=0.0000,14035.5909
EC01826=0.0000,14038.1201
EC01827=0.0000,14040.0000
EC01828=0.0000,14041.8799
EC01829=0.0000,14044.4091
EC01830=0.0000,14047.3837
EC01831=0.0000,14048.2508
EC01832=0.0000,14048.2514
EC01833=0.0000,14048.1286
EC01834=0.0000,14048.0287
EC01835=0.0000,14048.1105
EC01836=0.0000,14049.7738
EC01837=0.0000,14052.7052
EC01838=0.0000,14056.4001
EC01839=0.0000,14060.4362
EC01840=0.0000,14064.5637
EC01841=0.0000,14068.5997
EC01842=0.0000,14072.2952
EC01843=0.0000,14075.2262
EC01844=0.0000,14076.8889
EC01845=0.0000,14076.9711
EC01846=0.0000,14076.8716
EC01847=0.0000,14076.7487
EC01848=0.0000,14076.7500
EC01849=0.0000,14077.6160
EC01850=0.0000,14080.5914
EC01851=0.0000,14083.1202
EC01852=0.0000,14085.0000
EC01853=0.0000,14086.8791
EC01854=0.0000,14089.4092
EC01855=0.0000,14092.3840
EC01856=0.0000,14093.2500
EC01857=0.0000,14093.2513
EC01858=0.0000,14093.1284
EC01859=0.0000,14093.0289
EC01860=0.0000,14093.1111
EC01861=0.0000,14094.7738
EC01862=0.0000,14097.7048
EC01863=0.0000,14101.4003
EC01864=0.0000,14105.4363
EC01865=0.0000,14109.5638
EC01866=0.0000,14113.5999
EC01867=0.0000,14117.2948
EC01868=0.0000,14120.2262
EC01869=0.0000,14121.8895
EC01870=0.0000,14121.9713
EC01871=0.0000,14121.8714
EC01872=0.0000,14121.7486
EC01873=0.0000,14121.7492
EC01874=0.0000,14122.6163
EC01875=0.0000,14125.5909
EC01876=0.0000,14128.1201
EC01877=0.0000,14130.0000
EC01878=0.0000,14130.0000
EC01879=0.0000,14131.8104
EC01880=0.0000,14134.3168
EC01881=0.0000,14137.3110
EC01882=0.0000,14138.1459
EC01883=0.0000,14138.1209
EC01884=0.0000,14137.9932
EC01885=0.0000,14137.8955
EC01886=0.0000,14137.9733
EC01887=0.0000,14139.6504
EC01888=0.0000,14142.6088
EC01889=0.0000,14146.3398
EC01890=0.0000,14150.4161
EC01891=0.0000,14154.5839
EC01892=0.0000,14158.6599
EC01893=0.0000,14162.3913
EC01894=0.0000,14165.3500
EC01895=0.0000,14167.0265
EC01896=0.0000,14167.1043
EC01897=0.0000,14167.0066
EC01898=0.0000,14166.8795
EC01899=0.0000,14166.8537
EC01900=0.0000,14167.6887
EC01901=0.0000,14170.6829
EC01902=0.0000,14173.1899
EC01903=0.0000,14175.0000
EC01904=0.0000,14176.8101
EC01905=0.0000,14179.3178
EC01906=0.0000,14182.3119
EC01907=0.0000,14183.1463
EC01908=0.0000,14183.1205
EC01909=0.0000,14182.9934
EC01910=0.0000,14182.8957
EC01911=0.0000,14182.9735
EC01912=0.0000,14184.6500
EC01913=0.0000,14187.6087
EC01914=0.0000,14191.3401
EC01915=0.0000,14195.4161
EC01916=0.0000,14199.5839
EC01917=0.0000,14203.6602
EC01918=0.0000,14207.3912
EC01919=0.0000,14210.3496
EC01920=0.0000,14212.0267
EC01921=0.0000,14212.1045
EC01922=0.0000,14212.0068
EC01923=0.0000,14211.8791
EC01924=0.0000,14211.8541
EC01925=0.0000,14212.6890
EC01926=0.0000,14215.6832
EC01927=0.0000,14218.1896
EC01928=0.0000,14220.0000
EC01929=0.0000,14221.8094
EC01930=0.0000,14224.3178
EC01931=0.0000,14227.3110
EC01932=0.0000,14228.1459
EC01933=0.0000,14228.1209
EC01934=0.0000,14227.9932
EC01935=0.0000,14227.8955
EC01936=0.0000,14227.9733
EC01937=0.0000,14229.6504
EC01938=0.0000,14232.6088
EC01939=0.0000,14236.3398
EC01940=0.0000,14240.4161
EC01941=0.0000,14244.5839
EC01942=0.0000,14248.6599
EC01943=0.0000,14252.3913
EC01944=0.0000,14255.3500
EC01945=0.0000,14257.0265
EC01946=0.0000,14257.1043
EC01947=0.0000,14257.0066
EC01948=0.0000,14256.8795
EC01949=0.0000,14256.8537
EC01950=0.0000,14257.6887
EC01951=0.0000,14260.6829
EC01952=0.0000,14263.1899
EC01953=0.0000,14265.0000
EC01954=0.0000,14266.8101
EC01955=0.0000,14269.3178
EC01956=0.0000,14272.3119
EC01957=0.0000,14273.1463
EC01958=0.0000,14273.1205
EC01959=0.0000,14272.9934
EC01960=0.0000,14272.8957
EC01961=0.0000,14272.9735
EC01962=0.0000,14274.6500
EC01963=0.0000,14277.6087
EC01964=0.0000,14281.3401
EC01965=0.0000,14285.4161
EC01966=0.0000,14289.5839
EC01967=0.0000,14293.6602
EC01968=0.0000,14297.3912
EC01969=0.0000,14300.3496
EC01970=0.0000,14302.0267
EC01971=0.0000,14302.1045
EC01972=0.0000,14302.0068
EC01973=0.0000,14301.8791
EC01974=0.0000,14301.8541
EC01975=0.0000,14302.6890
EC01976=0.0000,14305.6832
EC01977=0.0000,14308.1896
EC01978=0.0000,14310.0000
EC01979=0.0000,14310.0000
EC01980=0.0000,14311.8094
EC01981=0.0000,14314.3178
EC01982=0.0000,14317.3110
EC01983=0.0000,14318.1459
EC01984=0.0000,14318.1209
EC01985=0.0000,14317.9932
EC01986=0.0000,14317.8955
EC01987=0.0000,14317.9733
EC01988=0.0000,14319.6504
EC01989=0.0000,14322.6088
EC01990=0.0000,14326.3398
EC01991=0.0000,14330.4161
EC01992=0.0000,14334.5839
EC01993=0.0000,14338.6599
EC01994=0.0000,14342.3913
EC01995=0.0000,14345.3500
EC01996=0.0000,14347.0265
EC01997=0.0000,14347.1043
EC01998=0.0000,14347.0066
EC01999=0.0000,14346.8795
//INST
///DATE 2022/04/08 11:15
///COMM
///ATTR SC,RW,RJ
////FRAME USER 2
///GROUP1 RB1
///GROUP2 ST1
NOP
SMOVL C00000 +MOVJ EC00000
SMOVL C00001 +MOVJ EC00001
SMOVL C00002 +MOVJ EC00002
SMOVL C00003 +MOVJ EC00003
SMOVL C00004 +MOVJ EC00004
SMOVL C00005 +MOVJ EC00005
SMOVL C00006 +MOVJ EC00006
SMOVL C00007 +MOVJ EC00007
SMOVL C00008 +MOVJ EC00008
SMOVL C00009 +MOVJ EC00009
SMOVL C00010 +MOVJ EC00010
SMOVL C00011 +MOVJ EC00011
SMOVL C00012 +MOVJ EC00012
SMOVL C00013 +MOVJ EC00013
SMOVL C00014 +MOVJ EC00014
SMOVL C00015 +MOVJ EC00015
SMOVL C00016 +MOVJ EC00016
SMOVL C00017 +MOVJ EC00017
SMOVL C00018 +MOVJ EC00018
SMOVL C00019 +MOVJ EC00019
SMOVL C00020 +MOVJ EC00020
SMOVL C00021 +MOVJ EC00021
SMOVL C00022 +MOVJ EC00022
SMOVL C00023 +MOVJ EC00023
SMOVL C00024 +MOVJ EC00024
SMOVL C00025 +MOVJ EC00025
SMOVL C00026 +MOVJ EC00026
SMOVL C00027 +MOVJ EC00027
SMOVL C00028 +MOVJ EC00028
SMOVL C00029 +MOVJ EC00029
SMOVL C00030 +MOVJ EC00030
SMOVL C00031 +MOVJ EC00031
SMOVL C00032 +MOVJ EC00032
SMOVL C00033 +MOVJ EC00033
SMOVL C00034 +MOVJ EC00034
SMOVL C00035 +MOVJ EC00035
SMOVL C00036 +MOVJ EC00036
SMOVL C00037 +MOVJ EC00037
SMOVL C00038 +MOVJ EC00038
SMOVL C00039 +MOVJ EC00039
SMOVL C00040 +MOVJ EC00040
SMOVL C00041 +MOVJ EC00041
SMOVL C00042 +MOVJ EC00042
SMOVL C00043 +MOVJ EC00043
SMOVL C00044 +MOVJ EC00044
SMOVL C00045 +MOVJ EC00045
SMOVL C00046 +MOVJ EC00046
SMOVL C00047 +MOVJ EC00047
SMOVL C00048 +MOVJ EC00048
SMOVL C00049 +MOVJ EC00049
SMOVL C00050 +MOVJ EC00050
SMOVL C00051 +MOVJ EC00051
SMOVL C00052 +MOVJ EC00052
SMOVL C00053 +MOVJ EC00053
SMOVL C00054 +MOVJ EC00054
SMOVL C00055 +MOVJ EC00055
SMOVL C00056 +MOVJ EC00056
SMOVL C00057 +MOVJ EC00057
SMOVL C00058 +MOVJ EC00058
SMOVL C00059 +MOVJ EC00059
SMOVL C00060 +MOVJ EC00060
SMOVL C00061 +MOVJ EC00061
SMOVL C00062 +MOVJ EC00062
SMOVL C00063 +MOVJ EC00063
SMOVL C00064 +MOVJ EC00064
SMOVL C00065 +MOVJ EC00065
SMOVL C00066 +MOVJ EC00066
SMOVL C00067 +MOVJ EC00067
SMOVL C00068 +MOVJ EC00068
SMOVL C00069 +MOVJ EC00069
SMOVL C00070 +MOVJ EC00070
SMOVL C00071 +MOVJ EC00071
SMOVL C00072 +MOVJ EC00072
SMOVL C00073 +MOVJ EC00073
SMOVL C00074 +MOVJ EC00074
SMOVL C00075 +MOVJ EC00075
SMOVL C00076 +MOVJ EC00076
SMOVL C00077 +MOVJ EC00077
SMOVL C00078 +MOVJ EC00078
SMOVL C00079 +MOVJ EC00079
SMOVL C00080 +MOVJ EC00080
SMOVL C00081 +MOVJ EC00081
SMOVL C00082 +MOVJ EC00082
SMOVL C00083 +MOVJ EC00083
SMOVL C00084 +MOVJ EC00084
SMOVL C00085 +MOVJ EC00085
SMOVL C00086 +MOVJ EC00086
SMOVL C00087 +MOVJ EC00087
SMOVL C00088 +MOVJ EC00088
SMOVL C00089 +MOVJ EC00089
SMOVL C00090 +MOVJ EC00090
SMOVL C00091 +MOVJ EC00091
SMOVL C00092 +MOVJ EC00092
SMOVL C00093 +MOVJ EC00093
SMOVL C00094 +MOVJ EC00094
SMOVL C00095 +MOVJ EC00095
SMOVL C00096 +MOVJ EC00096
SMOVL C00097 +MOVJ EC00097
SMOVL C00098 +MOVJ EC00098
SMOVL C00099 +MOVJ EC00099
SMOVL C00100 +MOVJ EC00100
SMOVL C00101 +MOVJ EC00101
SMOVL C00102 +MOVJ EC00102
SMOVL C00103 +MOVJ EC00103
SMOVL C00104 +MOVJ EC00104
SMOVL C00105 +MOVJ EC00105
SMOVL C00106 +MOVJ EC00106
SMOVL C00107 +MOVJ EC00107
SMOVL C00108 +MOVJ EC00108
SMOVL C00109 +MOVJ EC00109
SMOVL C00110 +MOVJ EC00110
SMOVL C00111 +MOVJ EC00111
SMOVL C00112 +MOVJ EC00112
SMOVL C00113 +MOVJ EC00113
SMOVL C00114 +MOVJ EC00114
SMOVL C00115 +MOVJ EC00115
SMOVL C00116 +MOVJ EC00116
SMOVL C00117 +MOVJ EC00117
SMOVL C00118 +MOVJ EC00118
SMOVL C00119 +MOVJ EC00119
SMOVL C00120 +MOVJ EC00120
SMOVL C00121 +MOVJ EC00121
SMOVL C00122 +MOVJ EC00122
SMOVL C00123 +MOVJ EC00123
SMOVL C00124 +MOVJ EC00124
SMOVL C00125 +MOVJ EC00125
SMOVL C00126 +MOVJ EC00126
SMOVL C00127 +MOVJ EC00127
SMOVL C00128 +MOVJ EC00128
SMOVL C00129 +MOVJ EC00129
SMOVL C00130 +MOVJ EC00130
SMOVL C00131 +MOVJ EC00131
SMOVL C00132 +MOVJ EC00132
SMOVL C00133 +MOVJ EC00133
SMOVL C00134 +MOVJ EC00134
SMOVL C00135 +MOVJ EC00135
SMOVL C00136 +MOVJ EC00136
SMOVL C00137 +MOVJ EC00137
SMOVL C00138 +MOVJ EC00138
SMOVL C00139 +MOVJ EC00139
SMOVL C00140 +MOVJ EC00140
SMOVL C00141 +MOVJ EC00141
SMOVL C00142 +MOVJ EC00142
SMOVL C00143 +MOVJ EC00143
SMOVL C00144 +MOVJ EC00144
SMOVL C00145 +MOVJ EC00145
SMOVL C00146 +MOVJ EC00146
SMOVL C00147 +MOVJ EC00147
SMOVL C00148 +MOVJ EC00148
SMOVL C00149 +MOVJ EC00149
SMOVL C00150 +MOVJ EC00150
SMOVL C00151 +MOVJ EC00151
SMOVL C00152 +MOVJ EC00152
SMOVL C00153 +MOVJ EC00153
SMOVL C00154 +MOVJ EC00154
SMOVL C00155 +MOVJ EC00155
SMOVL C00156 +MOVJ EC00156
SMOVL C00157 +MOVJ EC00157
SMOVL C00158 +MOVJ EC00158
SMOVL C00159 +MOVJ EC00159
SMOVL C00160 +MOVJ EC00160
SMOVL C00161 +MOVJ EC00161
SMOVL C00162 +MOVJ EC00162
SMOVL C00163 +MOVJ EC00163
SMOVL C00164 +MOVJ EC00164
SMOVL C00165 +MOVJ EC00165
SMOVL C00166 +MOVJ EC00166
SMOVL C00167 +MOVJ EC00167
SMOVL C00168 +MOVJ EC00168
SMOVL C00169 +MOVJ EC00169
SMOVL C00170 +MOVJ EC00170
SMOVL C00171 +MOVJ EC00171
SMOVL C00172 +MOVJ EC00172
SMOVL C00173 +MOVJ EC00173
SMOVL C00174 +MOVJ EC00174
SMOVL C00175 +MOVJ EC00175
SMOVL C00176 +MOVJ EC00176
SMOVL C00177 +MOVJ EC00177
SMOVL C00178 +MOVJ EC00178
SMOVL C00179 +MOVJ EC00179
SMOVL C00180 +MOVJ EC00180
SMOVL C00181 +MOVJ EC00181
SMOVL C00182 +MOVJ EC00182
SMOVL C00183 +MOVJ EC00183
SMOVL C00184 +MOVJ EC00184
SMOVL C00185 +MOVJ EC00185
SMOVL C00186 +MOVJ EC00186
SMOVL C00187 +MOVJ EC00187
SMOVL C00188 +MOVJ EC00188
SMOVL C00189 +MOVJ EC00189
SMOVL C00190 +MOVJ EC00190
SMOVL C00191 +MOVJ EC00191
SMOVL C00192 +MOVJ EC00192
SMOVL C00193 +MOVJ EC00193
SMOVL C00194 +MOVJ EC00194
SMOVL C00195 +MOVJ EC00195
SMOVL C00196 +MOVJ EC00196
SMOVL C00197 +MOVJ EC00197
SMOVL C00198 +MOVJ EC00198
SMOVL C00199 +MOVJ EC00199
SMOVL C00200 +MOVJ EC00200
SMOVL C00201 +MOVJ EC00201
SMOVL C00202 +MOVJ EC00202
SMOVL C00203 +MOVJ EC00203
SMOVL C00204 +MOVJ EC00204
SMOVL C00205 +MOVJ EC00205
SMOVL C00206 +MOVJ EC00206
SMOVL C00207 +MOVJ EC00207
SMOVL C00208 +MOVJ EC00208
SMOVL C00209 +MOVJ EC00209
SMOVL C00210 +MOVJ EC00210
SMOVL C00211 +MOVJ EC00211
SMOVL C00212 +MOVJ EC00212
SMOVL C00213 +MOVJ EC00213
SMOVL C00214 +MOVJ EC00214
SMOVL C00215 +MOVJ EC00215
SMOVL C00216 +MOVJ EC00216
SMOVL C00217 +MOVJ EC00217
SMOVL C00218 +MOVJ EC00218
SMOVL C00219 +MOVJ EC00219
SMOVL C00220 +MOVJ EC00220
SMOVL C00221 +MOVJ EC00221
SMOVL C00222 +MOVJ EC00222
SMOVL C00223 +MOVJ EC00223
SMOVL C00224 +MOVJ EC00224
SMOVL C00225 +MOVJ EC00225
SMOVL C00226 +MOVJ EC00226
SMOVL C00227 +MOVJ EC00227
SMOVL C00228 +MOVJ EC00228
SMOVL C00229 +MOVJ EC00229
SMOVL C00230 +MOVJ EC00230
SMOVL C00231 +MOVJ EC00231
SMOVL C00232 +MOVJ EC00232
SMOVL C00233 +MOVJ EC00233
SMOVL C00234 +MOVJ EC00234
SMOVL C00235 +MOVJ EC00235
SMOVL C00236 +MOVJ EC00236
SMOVL C00237 +MOVJ EC00237
SMOVL C00238 +MOVJ EC00238
SMOVL C00239 +MOVJ EC00239
SMOVL C00240 +MOVJ EC00240
SMOVL C00241 +MOVJ EC00241
SMOVL C00242 +MOVJ EC00242
SMOVL C00243 +MOVJ EC00243
SMOVL C00244 +MOVJ EC00244
SMOVL C00245 +MOVJ EC00245
SMOVL C00246 +MOVJ EC00246
SMOVL C00247 +MOVJ EC00247
SMOVL C00248 +MOVJ EC00248
SMOVL C00249 +MOVJ EC00249
SMOVL C00250 +MOVJ EC00250
SMOVL C00251 +MOVJ EC00251
SMOVL C00252 +MOVJ EC00252
SMOVL C00253 +MOVJ EC00253
SMOVL C00254 +MOVJ EC00254
SMOVL C00255 +MOVJ EC00255
SMOVL C00256 +MOVJ EC00256
SMOVL C00257 +MOVJ EC00257
SMOVL C00258 +MOVJ EC00258
SMOVL C00259 +MOVJ EC00259
SMOVL C00260 +MOVJ EC00260
SMOVL C00261 +MOVJ EC00261
SMOVL C00262 +MOVJ EC00262
SMOVL C00263 +MOVJ EC00263
SMOVL C00264 +MOVJ EC00264
SMOVL C00265 +MOVJ EC00265
SMOVL C00266 +MOVJ EC00266
SMOVL C00267 +MOVJ EC00267
SMOVL C00268 +MOVJ EC00268
SMOVL C00269 +MOVJ EC00269
SMOVL C00270 +MOVJ EC00270
SMOVL C00271 +MOVJ EC00271
SMOVL C00272 +MOVJ EC00272
SMOVL C00273 +MOVJ EC00273
SMOVL C00274 +MOVJ EC00274
SMOVL C00275 +MOVJ EC00275
SMOVL C00276 +MOVJ EC00276
SMOVL C00277 +MOVJ EC00277
SMOVL C00278 +MOVJ EC00278
SMOVL C00279 +MOVJ EC00279
SMOVL C00280 +MOVJ EC00280
SMOVL C00281 +MOVJ EC00281
SMOVL C00282 +MOVJ EC00282
SMOVL C00283 +MOVJ EC00283
SMOVL C00284 +MOVJ EC00284
SMOVL C00285 +MOVJ EC00285
SMOVL C00286 +MOVJ EC00286
SMOVL C00287 +MOVJ EC00287
SMOVL C00288 +MOVJ EC00288
SMOVL C00289 +MOVJ EC00289
SMOVL C00290 +MOVJ EC00290
SMOVL C00291 +MOVJ EC00291
SMOVL C00292 +MOVJ EC00292
SMOVL C00293 +MOVJ EC00293
SMOVL C00294 +MOVJ EC00294
SMOVL C00295 +MOVJ EC00295
SMOVL C00296 +MOVJ EC00296
SMOVL C00297 +MOVJ EC00297
SMOVL C00298 +MOVJ EC00298
SMOVL C00299 +MOVJ EC00299
SMOVL C00300 +MOVJ EC00300
SMOVL C00301 +MOVJ EC00301
SMOVL C00302 +MOVJ EC00302
SMOVL C00303 +MOVJ EC00303
SMOVL C00304 +MOVJ EC00304
SMOVL C00305 +MOVJ EC00305
SMOVL C00306 +MOVJ EC00306
SMOVL C00307 +MOVJ EC00307
SMOVL C00308 +MOVJ EC00308
SMOVL C00309 +MOVJ EC00309
SMOVL C00310 +MOVJ EC00310
SMOVL C00311 +MOVJ EC00311
SMOVL C00312 +MOVJ EC00312
SMOVL C00313 +MOVJ EC00313
SMOVL C00314 +MOVJ EC00314
SMOVL C00315 +MOVJ EC00315
SMOVL C00316 +MOVJ EC00316
SMOVL C00317 +MOVJ EC00317
SMOVL C00318 +MOVJ EC00318
SMOVL C00319 +MOVJ EC00319
SMOVL C00320 +MOVJ EC00320
SMOVL C00321 +MOVJ EC00321
SMOVL C00322 +MOVJ EC00322
SMOVL C00323 +MOVJ EC00323
SMOVL C00324 +MOVJ EC00324
SMOVL C00325 +MOVJ EC00325
SMOVL C00326 +MOVJ EC00326
SMOVL C00327 +MOVJ EC00327
SMOVL C00328 +MOVJ EC00328
SMOVL C00329 +MOVJ EC00329
SMOVL C00330 +MOVJ EC00330
SMOVL C00331 +MOVJ EC00331
SMOVL C00332 +MOVJ EC00332
SMOVL C00333 +MOVJ EC00333
SMOVL C00334 +MOVJ EC00334
SMOVL C00335 +MOVJ EC00335
SMOVL C00336 +MOVJ EC00336
SMOVL C00337 +MOVJ EC00337
SMOVL C00338 +MOVJ EC00338
SMOVL C00339 +MOVJ EC00339
SMOVL C00340 +MOVJ EC00340
SMOVL C00341 +MOVJ EC00341
SMOVL C00342 +MOVJ EC00342
SMOVL C00343 +MOVJ EC00343
SMOVL C00344 +MOVJ EC00344
SMOVL C00345 +MOVJ EC00345
SMOVL C00346 +MOVJ EC00346
SMOVL C00347 +MOVJ EC00347
SMOVL C00348 +MOVJ EC00348
SMOVL C00349 +MOVJ EC00349
SMOVL C00350 +MOVJ EC00350
SMOVL C00351 +MOVJ EC00351
SMOVL C00352 +MOVJ EC00352
SMOVL C00353 +MOVJ EC00353
SMOVL C00354 +MOVJ EC00354
SMOVL C00355 +MOVJ EC00355
SMOVL C00356 +MOVJ EC00356
SMOVL C00357 +MOVJ EC00357
SMOVL C00358 +MOVJ EC00358
SMOVL C00359 +MOVJ EC00359
SMOVL C00360 +MOVJ EC00360
SMOVL C00361 +MOVJ EC00361
SMOVL C00362 +MOVJ EC00362
SMOVL C00363 +MOVJ EC00363
SMOVL C00364 +MOVJ EC00364
SMOVL C00365 +MOVJ EC00365
SMOVL C00366 +MOVJ EC00366
SMOVL C00367 +MOVJ EC00367
SMOVL C00368 +MOVJ EC00368
SMOVL C00369 +MOVJ EC00369
SMOVL C00370 +MOVJ EC00370
SMOVL C00371 +MOVJ EC00371
SMOVL C00372 +MOVJ EC00372
SMOVL C00373 +MOVJ EC00373
SMOVL C00374 +MOVJ EC00374
SMOVL C00375 +MOVJ EC00375
SMOVL C00376 +MOVJ EC00376
SMOVL C00377 +MOVJ EC00377
SMOVL C00378 +MOVJ EC00378
SMOVL C00379 +MOVJ EC00379
SMOVL C00380 +MOVJ EC00380
SMOVL C00381 +MOVJ EC00381
SMOVL C00382 +MOVJ EC00382
SMOVL C00383 +MOVJ EC00383
SMOVL C00384 +MOVJ EC00384
SMOVL C00385 +MOVJ EC00385
SMOVL C00386 +MOVJ EC00386
SMOVL C00387 +MOVJ EC00387
SMOVL C00388 +MOVJ EC00388
SMOVL C00389 +MOVJ EC00389
SMOVL C00390 +MOVJ EC00390
SMOVL C00391 +MOVJ EC00391
SMOVL C00392 +MOVJ EC00392
SMOVL C00393 +MOVJ EC00393
SMOVL C00394 +MOVJ EC00394
SMOVL C00395 +MOVJ EC00395
SMOVL C00396 +MOVJ EC00396
SMOVL C00397 +MOVJ EC00397
SMOVL C00398 +MOVJ EC00398
SMOVL C00399 +MOVJ EC00399
SMOVL C00400 +MOVJ EC00400
SMOVL C00401 +MOVJ EC00401
SMOVL C00402 +MOVJ EC00402
SMOVL C00403 +MOVJ EC00403
SMOVL C00404 +MOVJ EC00404
SMOVL C00405 +MOVJ EC00405
SMOVL C00406 +MOVJ EC00406
SMOVL C00407 +MOVJ EC00407
SMOVL C00408 +MOVJ EC00408
SMOVL C00409 +MOVJ EC00409
SMOVL C00410 +MOVJ EC00410
SMOVL C00411 +MOVJ EC00411
SMOVL C00412 +MOVJ EC00412
SMOVL C00413 +MOVJ EC00413
SMOVL C00414 +MOVJ EC00414
SMOVL C00415 +MOVJ EC00415
SMOVL C00416 +MOVJ EC00416
SMOVL C00417 +MOVJ EC00417
SMOVL C00418 +MOVJ EC00418
SMOVL C00419 +MOVJ EC00419
SMOVL C00420 +MOVJ EC00420
SMOVL C00421 +MOVJ EC00421
SMOVL C00422 +MOVJ EC00422
SMOVL C00423 +MOVJ EC00423
SMOVL C00424 +MOVJ EC00424
SMOVL C00425 +MOVJ EC00425
SMOVL C00426 +MOVJ EC00426
SMOVL C00427 +MOVJ EC00427
SMOVL C00428 +MOVJ EC00428
SMOVL C00429 +MOVJ EC00429
SMOVL C00430 +MOVJ EC00430
SMOVL C00431 +MOVJ EC00431
SMOVL C00432 +MOVJ EC00432
SMOVL C00433 +MOVJ EC00433
SMOVL C00434 +MOVJ EC00434
SMOVL C00435 +MOVJ EC00435
SMOVL C00436 +MOVJ EC00436
SMOVL C00437 +MOVJ EC00437
SMOVL C00438 +MOVJ EC00438
SMOVL C00439 +MOVJ EC00439
SMOVL C00440 +MOVJ EC00440
SMOVL C00441 +MOVJ EC00441
SMOVL C00442 +MOVJ EC00442
SMOVL C00443 +MOVJ EC00443
SMOVL C00444 +MOVJ EC00444
SMOVL C00445 +MOVJ EC00445
SMOVL C00446 +MOVJ EC00446
SMOVL C00447 +MOVJ EC00447
SMOVL C00448 +MOVJ EC00448
SMOVL C00449 +MOVJ EC00449
SMOVL C00450 +MOVJ EC00450
SMOVL C00451 +MOVJ EC00451
SMOVL C00452 +MOVJ EC00452
SMOVL C00453 +MOVJ EC00453
SMOVL C00454 +MOVJ EC00454
SMOVL C00455 +MOVJ EC00455
SMOVL C00456 +MOVJ EC00456
SMOVL C00457 +MOVJ EC00457
SMOVL C00458 +MOVJ EC00458
SMOVL C00459 +MOVJ EC00459
SMOVL C00460 +MOVJ EC00460
SMOVL C00461 +MOVJ EC00461
SMOVL C00462 +MOVJ EC00462
SMOVL C00463 +MOVJ EC00463
SMOVL C00464 +MOVJ EC00464
SMOVL C00465 +MOVJ EC00465
SMOVL C00466 +MOVJ EC00466
SMOVL C00467 +MOVJ EC00467
SMOVL C00468 +MOVJ EC00468
SMOVL C00469 +MOVJ EC00469
SMOVL C00470 +MOVJ EC00470
SMOVL C00471 +MOVJ EC00471
SMOVL C00472 +MOVJ EC00472
SMOVL C00473 +MOVJ EC00473
SMOVL C00474 +MOVJ EC00474
SMOVL C00475 +MOVJ EC00475
SMOVL C00476 +MOVJ EC00476
SMOVL C00477 +MOVJ EC00477
SMOVL C00478 +MOVJ EC00478
SMOVL C00479 +MOVJ EC00479
SMOVL C00480 +MOVJ EC00480
SMOVL C00481 +MOVJ EC00481
SMOVL C00482 +MOVJ EC00482
SMOVL C00483 +MOVJ EC00483
SMOVL C00484 +MOVJ EC00484
SMOVL C00485 +MOVJ EC00485
SMOVL C00486 +MOVJ EC00486
SMOVL C00487 +MOVJ EC00487
SMOVL C00488 +MOVJ EC00488
SMOVL C00489 +MOVJ EC00489
SMOVL C00490 +MOVJ EC00490
SMOVL C00491 +MOVJ EC00491
SMOVL C00492 +MOVJ EC00492
SMOVL C00493 +MOVJ EC00493
SMOVL C00494 +MOVJ EC00494
SMOVL C00495 +MOVJ EC00495
SMOVL C00496 +MOVJ EC00496
SMOVL C00497 +MOVJ EC00497
SMOVL C00498 +MOVJ EC00498
SMOVL C00499 +MOVJ EC00499
SMOVL C00500 +MOVJ EC00500
SMOVL C00501 +MOVJ EC00501
SMOVL C00502 +MOVJ EC00502
SMOVL C00503 +MOVJ EC00503
SMOVL C00504 +MOVJ EC00504
SMOVL C00505 +MOVJ EC00505
SMOVL C00506 +MOVJ EC00506
SMOVL C00507 +MOVJ EC00507
SMOVL C00508 +MOVJ EC00508
SMOVL C00509 +MOVJ EC00509
SMOVL C00510 +MOVJ EC00510
SMOVL C00511 +MOVJ EC00511
SMOVL C00512 +MOVJ EC00512
SMOVL C00513 +MOVJ EC00513
SMOVL C00514 +MOVJ EC00514
SMOVL C00515 +MOVJ EC00515
SMOVL C00516 +MOVJ EC00516
SMOVL C00517 +MOVJ EC00517
SMOVL C00518 +MOVJ EC00518
SMOVL C00519 +MOVJ EC00519
SMOVL C00520 +MOVJ EC00520
SMOVL C00521 +MOVJ EC00521
SMOVL C00522 +MOVJ EC00522
SMOVL C00523 +MOVJ EC00523
SMOVL C00524 +MOVJ EC00524
SMOVL C00525 +MOVJ EC00525
SMOVL C00526 +MOVJ EC00526
SMOVL C00527 +MOVJ EC00527
SMOVL C00528 +MOVJ EC00528
SMOVL C00529 +MOVJ EC00529
SMOVL C00530 +MOVJ EC00530
SMOVL C00531 +MOVJ EC00531
SMOVL C00532 +MOVJ EC00532
SMOVL C00533 +MOVJ EC00533
SMOVL C00534 +MOVJ EC00534
SMOVL C00535 +MOVJ EC00535
SMOVL C00536 +MOVJ EC00536
SMOVL C00537 +MOVJ EC00537
SMOVL C00538 +MOVJ EC00538
SMOVL C00539 +MOVJ EC00539
SMOVL C00540 +MOVJ EC00540
SMOVL C00541 +MOVJ EC00541
SMOVL C00542 +MOVJ EC00542
SMOVL C00543 +MOVJ EC00543
SMOVL C00544 +MOVJ EC00544
SMOVL C00545 +MOVJ EC00545
SMOVL C00546 +MOVJ EC00546
SMOVL C00547 +MOVJ EC00547
SMOVL C00548 +MOVJ EC00548
SMOVL C00549 +MOVJ EC00549
SMOVL C00550 +MOVJ EC00550
SMOVL C00551 +MOVJ EC00551
SMOVL C00552 +MOVJ EC00552
SMOVL C00553 +MOVJ EC00553
SMOVL C00554 +MOVJ EC00554
SMOVL C00555 +MOVJ EC00555
SMOVL C00556 +MOVJ EC00556
SMOVL C00557 +MOVJ EC00557
SMOVL C00558 +MOVJ EC00558
SMOVL C00559 +MOVJ EC00559
SMOVL C00560 +MOVJ EC00560
SMOVL C00561 +MOVJ EC00561
SMOVL C00562 +MOVJ EC00562
SMOVL C00563 +MOVJ EC00563
SMOVL C00564 +MOVJ EC00564
SMOVL C00565 +MOVJ EC00565
SMOVL C00566 +MOVJ EC00566
SMOVL C00567 +MOVJ EC00567
SMOVL C00568 +MOVJ EC00568
SMOVL C00569 +MOVJ EC00569
SMOVL C00570 +MOVJ EC00570
SMOVL C00571 +MOVJ EC00571
SMOVL C00572 +MOVJ EC00572
SMOVL C00573 +MOVJ EC00573
SMOVL C00574 +MOVJ EC00574
SMOVL C00575 +MOVJ EC00575
SMOVL C00576 +MOVJ EC00576
SMOVL C00577 +MOVJ EC00577
SMOVL C00578 +MOVJ EC00578
SMOVL C00579 +MOVJ EC00579
SMOVL C00580 +MOVJ EC00580
SMOVL C00581 +MOVJ EC00581
SMOVL C00582 +MOVJ EC00582
SMOVL C00583 +MOVJ EC00583
SMOVL C00584 +MOVJ EC00584
SMOVL C00585 +MOVJ EC00585
SMOVL C00586 +MOVJ EC00586
SMOVL C00587 +MOVJ EC00587
SMOVL C00588 +MOVJ EC00588
SMOVL C00589 +MOVJ EC00589
SMOVL C00590 +MOVJ EC00590
SMOVL C00591 +MOVJ EC00591
SMOVL C00592 +MOVJ EC00592
SMOVL C00593 +MOVJ EC00593
SMOVL C00594 +MOVJ EC00594
SMOVL C00595 +MOVJ EC00595
SMOVL C00596 +MOVJ EC00596
SMOVL C00597 +MOVJ EC00597
SMOVL C00598 +MOVJ EC00598
SMOVL C00599 +MOVJ EC00599
SMOVL C00600 +MOVJ EC00600
SMOVL C00601 +MOVJ EC00601
SMOVL C00602 +MOVJ EC00602
SMOVL C00603 +MOVJ EC00603
SMOVL C00604 +MOVJ EC00604
SMOVL C00605 +MOVJ EC00605
SMOVL C00606 +MOVJ EC00606
SMOVL C00607 +MOVJ EC00607
SMOVL C00608 +MOVJ EC00608
SMOVL C00609 +MOVJ EC00609
SMOVL C00610 +MOVJ EC00610
SMOVL C00611 +MOVJ EC00611
SMOVL C00612 +MOVJ EC00612
SMOVL C00613 +MOVJ EC00613
SMOVL C00614 +MOVJ EC00614
SMOVL C00615 +MOVJ EC00615
SMOVL C00616 +MOVJ EC00616
SMOVL C00617 +MOVJ EC00617
SMOVL C00618 +MOVJ EC00618
SMOVL C00619 +MOVJ EC00619
SMOVL C00620 +MOVJ EC00620
SMOVL C00621 +MOVJ EC00621
SMOVL C00622 +MOVJ EC00622
SMOVL C00623 +MOVJ EC00623
SMOVL C00624 +MOVJ EC00624
SMOVL C00625 +MOVJ EC00625
SMOVL C00626 +MOVJ EC00626
SMOVL C00627 +MOVJ EC00627
SMOVL C00628 +MOVJ EC00628
SMOVL C00629 +MOVJ EC00629
SMOVL C00630 +MOVJ EC00630
SMOVL C00631 +MOVJ EC00631
SMOVL C00632 +MOVJ EC00632
SMOVL C00633 +MOVJ EC00633
SMOVL C00634 +MOVJ EC00634
SMOVL C00635 +MOVJ EC00635
SMOVL C00636 +MOVJ EC00636
SMOVL C00637 +MOVJ EC00637
SMOVL C00638 +MOVJ EC00638
SMOVL C00639 +MOVJ EC00639
SMOVL C00640 +MOVJ EC00640
SMOVL C00641 +MOVJ EC00641
SMOVL C00642 +MOVJ EC00642
SMOVL C00643 +MOVJ EC00643
SMOVL C00644 +MOVJ EC00644
SMOVL C00645 +MOVJ EC00645
SMOVL C00646 +MOVJ EC00646
SMOVL C00647 +MOVJ EC00647
SMOVL C00648 +MOVJ EC00648
SMOVL C00649 +MOVJ EC00649
SMOVL C00650 +MOVJ EC00650
SMOVL C00651 +MOVJ EC00651
SMOVL C00652 +MOVJ EC00652
SMOVL C00653 +MOVJ EC00653
SMOVL C00654 +MOVJ EC00654
SMOVL C00655 +MOVJ EC00655
SMOVL C00656 +MOVJ EC00656
SMOVL C00657 +MOVJ EC00657
SMOVL C00658 +MOVJ EC00658
SMOVL C00659 +MOVJ EC00659
SMOVL C00660 +MOVJ EC00660
SMOVL C00661 +MOVJ EC00661
SMOVL C00662 +MOVJ EC00662
SMOVL C00663 +MOVJ EC00663
SMOVL C00664 +MOVJ EC00664
SMOVL C00665 +MOVJ EC00665
SMOVL C00666 +MOVJ EC00666
SMOVL C00667 +MOVJ EC00667
SMOVL C00668 +MOVJ EC00668
SMOVL C00669 +MOVJ EC00669
SMOVL C00670 +MOVJ EC00670
SMOVL C00671 +MOVJ EC00671
SMOVL C00672 +MOVJ EC00672
SMOVL C00673 +MOVJ EC00673
SMOVL C00674 +MOVJ EC00674
SMOVL C00675 +MOVJ EC00675
SMOVL C00676 +MOVJ EC00676
SMOVL C00677 +MOVJ EC00677
SMOVL C00678 +MOVJ EC00678
SMOVL C00679 +MOVJ EC00679
SMOVL C00680 +MOVJ EC00680
SMOVL C00681 +MOVJ EC00681
SMOVL C00682 +MOVJ EC00682
SMOVL C00683 +MOVJ EC00683
SMOVL C00684 +MOVJ EC00684
SMOVL C00685 +MOVJ EC00685
SMOVL C00686 +MOVJ EC00686
SMOVL C00687 +MOVJ EC00687
SMOVL C00688 +MOVJ EC00688
SMOVL C00689 +MOVJ EC00689
SMOVL C00690 +MOVJ EC00690
SMOVL C00691 +MOVJ EC00691
SMOVL C00692 +MOVJ EC00692
SMOVL C00693 +MOVJ EC00693
SMOVL C00694 +MOVJ EC00694
SMOVL C00695 +MOVJ EC00695
SMOVL C00696 +MOVJ EC00696
SMOVL C00697 +MOVJ EC00697
SMOVL C00698 +MOVJ EC00698
SMOVL C00699 +MOVJ EC00699
SMOVL C00700 +MOVJ EC00700
SMOVL C00701 +MOVJ EC00701
SMOVL C00702 +MOVJ EC00702
SMOVL C00703 +MOVJ EC00703
SMOVL C00704 +MOVJ EC00704
SMOVL C00705 +MOVJ EC00705
SMOVL C00706 +MOVJ EC00706
SMOVL C00707 +MOVJ EC00707
SMOVL C00708 +MOVJ EC00708
SMOVL C00709 +MOVJ EC00709
SMOVL C00710 +MOVJ EC00710
SMOVL C00711 +MOVJ EC00711
SMOVL C00712 +MOVJ EC00712
SMOVL C00713 +MOVJ EC00713
SMOVL C00714 +MOVJ EC00714
SMOVL C00715 +MOVJ EC00715
SMOVL C00716 +MOVJ EC00716
SMOVL C00717 +MOVJ EC00717
SMOVL C00718 +MOVJ EC00718
SMOVL C00719 +MOVJ EC00719
SMOVL C00720 +MOVJ EC00720
SMOVL C00721 +MOVJ EC00721
SMOVL C00722 +MOVJ EC00722
SMOVL C00723 +MOVJ EC00723
SMOVL C00724 +MOVJ EC00724
SMOVL C00725 +MOVJ EC00725
SMOVL C00726 +MOVJ EC00726
SMOVL C00727 +MOVJ EC00727
SMOVL C00728 +MOVJ EC00728
SMOVL C00729 +MOVJ EC00729
SMOVL C00730 +MOVJ EC00730
SMOVL C00731 +MOVJ EC00731
SMOVL C00732 +MOVJ EC00732
SMOVL C00733 +MOVJ EC00733
SMOVL C00734 +MOVJ EC00734
SMOVL C00735 +MOVJ EC00735
SMOVL C00736 +MOVJ EC00736
SMOVL C00737 +MOVJ EC00737
SMOVL C00738 +MOVJ EC00738
SMOVL C00739 +MOVJ EC00739
SMOVL C00740 +MOVJ EC00740
SMOVL C00741 +MOVJ EC00741
SMOVL C00742 +MOVJ EC00742
SMOVL C00743 +MOVJ EC00743
SMOVL C00744 +MOVJ EC00744
SMOVL C00745 +MOVJ EC00745
SMOVL C00746 +MOVJ EC00746
SMOVL C00747 +MOVJ EC00747
SMOVL C00748 +MOVJ EC00748
SMOVL C00749 +MOVJ EC00749
SMOVL C00750 +MOVJ EC00750
SMOVL C00751 +MOVJ EC00751
SMOVL C00752 +MOVJ EC00752
SMOVL C00753 +MOVJ EC00753
SMOVL C00754 +MOVJ EC00754
SMOVL C00755 +MOVJ EC00755
SMOVL C00756 +MOVJ EC00756
SMOVL C00757 +MOVJ EC00757
SMOVL C00758 +MOVJ EC00758
SMOVL C00759 +MOVJ EC00759
SMOVL C00760 +MOVJ EC00760
SMOVL C00761 +MOVJ EC00761
SMOVL C00762 +MOVJ EC00762
SMOVL C00763 +MOVJ EC00763
SMOVL C00764 +MOVJ EC00764
SMOVL C00765 +MOVJ EC00765
SMOVL C00766 +MOVJ EC00766
SMOVL C00767 +MOVJ EC00767
SMOVL C00768 +MOVJ EC00768
SMOVL C00769 +MOVJ EC00769
SMOVL C00770 +MOVJ EC00770
SMOVL C00771 +MOVJ EC00771
SMOVL C00772 +MOVJ EC00772
SMOVL C00773 +MOVJ EC00773
SMOVL C00774 +MOVJ EC00774
SMOVL C00775 +MOVJ EC00775
SMOVL C00776 +MOVJ EC00776
SMOVL C00777 +MOVJ EC00777
SMOVL C00778 +MOVJ EC00778
SMOVL C00779 +MOVJ EC00779
SMOVL C00780 +MOVJ EC00780
SMOVL C00781 +MOVJ EC00781
SMOVL C00782 +MOVJ EC00782
SMOVL C00783 +MOVJ EC00783
SMOVL C00784 +MOVJ EC00784
SMOVL C00785 +MOVJ EC00785
SMOVL C00786 +MOVJ EC00786
SMOVL C00787 +MOVJ EC00787
SMOVL C00788 +MOVJ EC00788
SMOVL C00789 +MOVJ EC00789
SMOVL C00790 +MOVJ EC00790
SMOVL C00791 +MOVJ EC00791
SMOVL C00792 +MOVJ EC00792
SMOVL C00793 +MOVJ EC00793
SMOVL C00794 +MOVJ EC00794
SMOVL C00795 +MOVJ EC00795
SMOVL C00796 +MOVJ EC00796
SMOVL C00797 +MOVJ EC00797
SMOVL C00798 +MOVJ EC00798
SMOVL C00799 +MOVJ EC00799
SMOVL C00800 +MOVJ EC00800
SMOVL C00801 +MOVJ EC00801
SMOVL C00802 +MOVJ EC00802
SMOVL C00803 +MOVJ EC00803
SMOVL C00804 +MOVJ EC00804
SMOVL C00805 +MOVJ EC00805
SMOVL C00806 +MOVJ EC00806
SMOVL C00807 +MOVJ EC00807
SMOVL C00808 +MOVJ EC00808
SMOVL C00809 +MOVJ EC00809
SMOVL C00810 +MOVJ EC00810
SMOVL C00811 +MOVJ EC00811
SMOVL C00812 +MOVJ EC00812
SMOVL C00813 +MOVJ EC00813
SMOVL C00814 +MOVJ EC00814
SMOVL C00815 +MOVJ EC00815
SMOVL C00816 +MOVJ EC00816
SMOVL C00817 +MOVJ EC00817
SMOVL C00818 +MOVJ EC00818
SMOVL C00819 +MOVJ EC00819
SMOVL C00820 +MOVJ EC00820
SMOVL C00821 +MOVJ EC00821
SMOVL C00822 +MOVJ EC00822
SMOVL C00823 +MOVJ EC00823
SMOVL C00824 +MOVJ EC00824
SMOVL C00825 +MOVJ EC00825
SMOVL C00826 +MOVJ EC00826
SMOVL C00827 +MOVJ EC00827
SMOVL C00828 +MOVJ EC00828
SMOVL C00829 +MOVJ EC00829
SMOVL C00830 +MOVJ EC00830
SMOVL C00831 +MOVJ EC00831
SMOVL C00832 +MOVJ EC00832
SMOVL C00833 +MOVJ EC00833
SMOVL C00834 +MOVJ EC00834
SMOVL C00835 +MOVJ EC00835
SMOVL C00836 +MOVJ EC00836
SMOVL C00837 +MOVJ EC00837
SMOVL C00838 +MOVJ EC00838
SMOVL C00839 +MOVJ EC00839
SMOVL C00840 +MOVJ EC00840
SMOVL C00841 +MOVJ EC00841
SMOVL C00842 +MOVJ EC00842
SMOVL C00843 +MOVJ EC00843
SMOVL C00844 +MOVJ EC00844
SMOVL C00845 +MOVJ EC00845
SMOVL C00846 +MOVJ EC00846
SMOVL C00847 +MOVJ EC00847
SMOVL C00848 +MOVJ EC00848
SMOVL C00849 +MOVJ EC00849
SMOVL C00850 +MOVJ EC00850
SMOVL C00851 +MOVJ EC00851
SMOVL C00852 +MOVJ EC00852
SMOVL C00853 +MOVJ EC00853
SMOVL C00854 +MOVJ EC00854
SMOVL C00855 +MOVJ EC00855
SMOVL C00856 +MOVJ EC00856
SMOVL C00857 +MOVJ EC00857
SMOVL C00858 +MOVJ EC00858
SMOVL C00859 +MOVJ EC00859
SMOVL C00860 +MOVJ EC00860
SMOVL C00861 +MOVJ EC00861
SMOVL C00862 +MOVJ EC00862
SMOVL C00863 +MOVJ EC00863
SMOVL C00864 +MOVJ EC00864
SMOVL C00865 +MOVJ EC00865
SMOVL C00866 +MOVJ EC00866
SMOVL C00867 +MOVJ EC00867
SMOVL C00868 +MOVJ EC00868
SMOVL C00869 +MOVJ EC00869
SMOVL C00870 +MOVJ EC00870
SMOVL C00871 +MOVJ EC00871
SMOVL C00872 +MOVJ EC00872
SMOVL C00873 +MOVJ EC00873
SMOVL C00874 +MOVJ EC00874
SMOVL C00875 +MOVJ EC00875
SMOVL C00876 +MOVJ EC00876
SMOVL C00877 +MOVJ EC00877
SMOVL C00878 +MOVJ EC00878
SMOVL C00879 +MOVJ EC00879
SMOVL C00880 +MOVJ EC00880
SMOVL C00881 +MOVJ EC00881
SMOVL C00882 +MOVJ EC00882
SMOVL C00883 +MOVJ EC00883
SMOVL C00884 +MOVJ EC00884
SMOVL C00885 +MOVJ EC00885
SMOVL C00886 +MOVJ EC00886
SMOVL C00887 +MOVJ EC00887
SMOVL C00888 +MOVJ EC00888
SMOVL C00889 +MOVJ EC00889
SMOVL C00890 +MOVJ EC00890
SMOVL C00891 +MOVJ EC00891
SMOVL C00892 +MOVJ EC00892
SMOVL C00893 +MOVJ EC00893
SMOVL C00894 +MOVJ EC00894
SMOVL C00895 +MOVJ EC00895
SMOVL C00896 +MOVJ EC00896
SMOVL C00897 +MOVJ EC00897
SMOVL C00898 +MOVJ EC00898
SMOVL C00899 +MOVJ EC00899
SMOVL C00900 +MOVJ EC00900
SMOVL C00901 +MOVJ EC00901
SMOVL C00902 +MOVJ EC00902
SMOVL C00903 +MOVJ EC00903
SMOVL C00904 +MOVJ EC00904
SMOVL C00905 +MOVJ EC00905
SMOVL C00906 +MOVJ EC00906
SMOVL C00907 +MOVJ EC00907
SMOVL C00908 +MOVJ EC00908
SMOVL C00909 +MOVJ EC00909
SMOVL C00910 +MOVJ EC00910
SMOVL C00911 +MOVJ EC00911
SMOVL C00912 +MOVJ EC00912
SMOVL C00913 +MOVJ EC00913
SMOVL C00914 +MOVJ EC00914
SMOVL C00915 +MOVJ EC00915
SMOVL C00916 +MOVJ EC00916
SMOVL C00917 +MOVJ EC00917
SMOVL C00918 +MOVJ EC00918
SMOVL C00919 +MOVJ EC00919
SMOVL C00920 +MOVJ EC00920
SMOVL C00921 +MOVJ EC00921
SMOVL C00922 +MOVJ EC00922
SMOVL C00923 +MOVJ EC00923
SMOVL C00924 +MOVJ EC00924
SMOVL C00925 +MOVJ EC00925
SMOVL C00926 +MOVJ EC00926
SMOVL C00927 +MOVJ EC00927
SMOVL C00928 +MOVJ EC00928
SMOVL C00929 +MOVJ EC00929
SMOVL C00930 +MOVJ EC00930
SMOVL C00931 +MOVJ EC00931
SMOVL C00932 +MOVJ EC00932
SMOVL C00933 +MOVJ EC00933
SMOVL C00934 +MOVJ EC00934
SMOVL C00935 +MOVJ EC00935
SMOVL C00936 +MOVJ EC00936
SMOVL C00937 +MOVJ EC00937
SMOVL C00938 +MOVJ EC00938
SMOVL C00939 +MOVJ EC00939
SMOVL C00940 +MOVJ EC00940
SMOVL C00941 +MOVJ EC00941
SMOVL C00942 +MOVJ EC00942
SMOVL C00943 +MOVJ EC00943
SMOVL C00944 +MOVJ EC00944
SMOVL C00945 +MOVJ EC00945
SMOVL C00946 +MOVJ EC00946
SMOVL C00947 +MOVJ EC00947
SMOVL C00948 +MOVJ EC00948
SMOVL C00949 +MOVJ EC00949
SMOVL C00950 +MOVJ EC00950
SMOVL C00951 +MOVJ EC00951
SMOVL C00952 +MOVJ EC00952
SMOVL C00953 +MOVJ EC00953
SMOVL C00954 +MOVJ EC00954
SMOVL C00955 +MOVJ EC00955
SMOVL C00956 +MOVJ EC00956
SMOVL C00957 +MOVJ EC00957
SMOVL C00958 +MOVJ EC00958
SMOVL C00959 +MOVJ EC00959
SMOVL C00960 +MOVJ EC00960
SMOVL C00961 +MOVJ EC00961
SMOVL C00962 +MOVJ EC00962
SMOVL C00963 +MOVJ EC00963
SMOVL C00964 +MOVJ EC00964
SMOVL C00965 +MOVJ EC00965
SMOVL C00966 +MOVJ EC00966
SMOVL C00967 +MOVJ EC00967
SMOVL C00968 +MOVJ EC00968
SMOVL C00969 +MOVJ EC00969
SMOVL C00970 +MOVJ EC00970
SMOVL C00971 +MOVJ EC00971
SMOVL C00972 +MOVJ EC00972
SMOVL C00973 +MOVJ EC00973
SMOVL C00974 +MOVJ EC00974
SMOVL C00975 +MOVJ EC00975
SMOVL C00976 +MOVJ EC00976
SMOVL C00977 +MOVJ EC00977
SMOVL C00978 +MOVJ EC00978
SMOVL C00979 +MOVJ EC00979
SMOVL C00980 +MOVJ EC00980
SMOVL C00981 +MOVJ EC00981
SMOVL C00982 +MOVJ EC00982
SMOVL C00983 +MOVJ EC00983
SMOVL C00984 +MOVJ EC00984
SMOVL C00985 +MOVJ EC00985
SMOVL C00986 +MOVJ EC00986
SMOVL C00987 +MOVJ EC00987
SMOVL C00988 +MOVJ EC00988
SMOVL C00989 +MOVJ EC00989
SMOVL C00990 +MOVJ EC00990
SMOVL C00991 +MOVJ EC00991
SMOVL C00992 +MOVJ EC00992
SMOVL C00993 +MOVJ EC00993
SMOVL C00994 +MOVJ EC00994
SMOVL C00995 +MOVJ EC00995
SMOVL C00996 +MOVJ EC00996
SMOVL C00997 +MOVJ EC00997
SMOVL C00998 +MOVJ EC00998
SMOVL C00999 +MOVJ EC00999
SMOVL C01000 +MOVJ EC01000
SMOVL C01001 +MOVJ EC01001
SMOVL C01002 +MOVJ EC01002
SMOVL C01003 +MOVJ EC01003
SMOVL C01004 +MOVJ EC01004
SMOVL C01005 +MOVJ EC01005
SMOVL C01006 +MOVJ EC01006
SMOVL C01007 +MOVJ EC01007
SMOVL C01008 +MOVJ EC01008
SMOVL C01009 +MOVJ EC01009
SMOVL C01010 +MOVJ EC01010
SMOVL C01011 +MOVJ EC01011
SMOVL C01012 +MOVJ EC01012
SMOVL C01013 +MOVJ EC01013
SMOVL C01014 +MOVJ EC01014
SMOVL C01015 +MOVJ EC01015
SMOVL C01016 +MOVJ EC01016
SMOVL C01017 +MOVJ EC01017
SMOVL C01018 +MOVJ EC01018
SMOVL C01019 +MOVJ EC01019
SMOVL C01020 +MOVJ EC01020
SMOVL C01021 +MOVJ EC01021
SMOVL C01022 +MOVJ EC01022
SMOVL C01023 +MOVJ EC01023
SMOVL C01024 +MOVJ EC01024
SMOVL C01025 +MOVJ EC01025
SMOVL C01026 +MOVJ EC01026
SMOVL C01027 +MOVJ EC01027
SMOVL C01028 +MOVJ EC01028
SMOVL C01029 +MOVJ EC01029
SMOVL C01030 +MOVJ EC01030
SMOVL C01031 +MOVJ EC01031
SMOVL C01032 +MOVJ EC01032
SMOVL C01033 +MOVJ EC01033
SMOVL C01034 +MOVJ EC01034
SMOVL C01035 +MOVJ EC01035
SMOVL C01036 +MOVJ EC01036
SMOVL C01037 +MOVJ EC01037
SMOVL C01038 +MOVJ EC01038
SMOVL C01039 +MOVJ EC01039
SMOVL C01040 +MOVJ EC01040
SMOVL C01041 +MOVJ EC01041
SMOVL C01042 +MOVJ EC01042
SMOVL C01043 +MOVJ EC01043
SMOVL C01044 +MOVJ EC01044
SMOVL C01045 +MOVJ EC01045
SMOVL C01046 +MOVJ EC01046
SMOVL C01047 +MOVJ EC01047
SMOVL C01048 +MOVJ EC01048
SMOVL C01049 +MOVJ EC01049
SMOVL C01050 +MOVJ EC01050
SMOVL C01051 +MOVJ EC01051
SMOVL C01052 +MOVJ EC01052
SMOVL C01053 +MOVJ EC01053
SMOVL C01054 +MOVJ EC01054
SMOVL C01055 +MOVJ EC01055
SMOVL C01056 +MOVJ EC01056
SMOVL C01057 +MOVJ EC01057
SMOVL C01058 +MOVJ EC01058
SMOVL C01059 +MOVJ EC01059
SMOVL C01060 +MOVJ EC01060
SMOVL C01061 +MOVJ EC01061
SMOVL C01062 +MOVJ EC01062
SMOVL C01063 +MOVJ EC01063
SMOVL C01064 +MOVJ EC01064
SMOVL C01065 +MOVJ EC01065
SMOVL C01066 +MOVJ EC01066
SMOVL C01067 +MOVJ EC01067
SMOVL C01068 +MOVJ EC01068
SMOVL C01069 +MOVJ EC01069
SMOVL C01070 +MOVJ EC01070
SMOVL C01071 +MOVJ EC01071
SMOVL C01072 +MOVJ EC01072
SMOVL C01073 +MOVJ EC01073
SMOVL C01074 +MOVJ EC01074
SMOVL C01075 +MOVJ EC01075
SMOVL C01076 +MOVJ EC01076
SMOVL C01077 +MOVJ EC01077
SMOVL C01078 +MOVJ EC01078
SMOVL C01079 +MOVJ EC01079
SMOVL C01080 +MOVJ EC01080
SMOVL C01081 +MOVJ EC01081
SMOVL C01082 +MOVJ EC01082
SMOVL C01083 +MOVJ EC01083
SMOVL C01084 +MOVJ EC01084
SMOVL C01085 +MOVJ EC01085
SMOVL C01086 +MOVJ EC01086
SMOVL C01087 +MOVJ EC01087
SMOVL C01088 +MOVJ EC01088
SMOVL C01089 +MOVJ EC01089
SMOVL C01090 +MOVJ EC01090
SMOVL C01091 +MOVJ EC01091
SMOVL C01092 +MOVJ EC01092
SMOVL C01093 +MOVJ EC01093
SMOVL C01094 +MOVJ EC01094
SMOVL C01095 +MOVJ EC01095
SMOVL C01096 +MOVJ EC01096
SMOVL C01097 +MOVJ EC01097
SMOVL C01098 +MOVJ EC01098
SMOVL C01099 +MOVJ EC01099
SMOVL C01100 +MOVJ EC01100
SMOVL C01101 +MOVJ EC01101
SMOVL C01102 +MOVJ EC01102
SMOVL C01103 +MOVJ EC01103
SMOVL C01104 +MOVJ EC01104
SMOVL C01105 +MOVJ EC01105
SMOVL C01106 +MOVJ EC01106
SMOVL C01107 +MOVJ EC01107
SMOVL C01108 +MOVJ EC01108
SMOVL C01109 +MOVJ EC01109
SMOVL C01110 +MOVJ EC01110
SMOVL C01111 +MOVJ EC01111
SMOVL C01112 +MOVJ EC01112
SMOVL C01113 +MOVJ EC01113
SMOVL C01114 +MOVJ EC01114
SMOVL C01115 +MOVJ EC01115
SMOVL C01116 +MOVJ EC01116
SMOVL C01117 +MOVJ EC01117
SMOVL C01118 +MOVJ EC01118
SMOVL C01119 +MOVJ EC01119
SMOVL C01120 +MOVJ EC01120
SMOVL C01121 +MOVJ EC01121
SMOVL C01122 +MOVJ EC01122
SMOVL C01123 +MOVJ EC01123
SMOVL C01124 +MOVJ EC01124
SMOVL C01125 +MOVJ EC01125
SMOVL C01126 +MOVJ EC01126
SMOVL C01127 +MOVJ EC01127
SMOVL C01128 +MOVJ EC01128
SMOVL C01129 +MOVJ EC01129
SMOVL C01130 +MOVJ EC01130
SMOVL C01131 +MOVJ EC01131
SMOVL C01132 +MOVJ EC01132
SMOVL C01133 +MOVJ EC01133
SMOVL C01134 +MOVJ EC01134
SMOVL C01135 +MOVJ EC01135
SMOVL C01136 +MOVJ EC01136
SMOVL C01137 +MOVJ EC01137
SMOVL C01138 +MOVJ EC01138
SMOVL C01139 +MOVJ EC01139
SMOVL C01140 +MOVJ EC01140
SMOVL C01141 +MOVJ EC01141
SMOVL C01142 +MOVJ EC01142
SMOVL C01143 +MOVJ EC01143
